RoboDK station: palletizing test.rdk

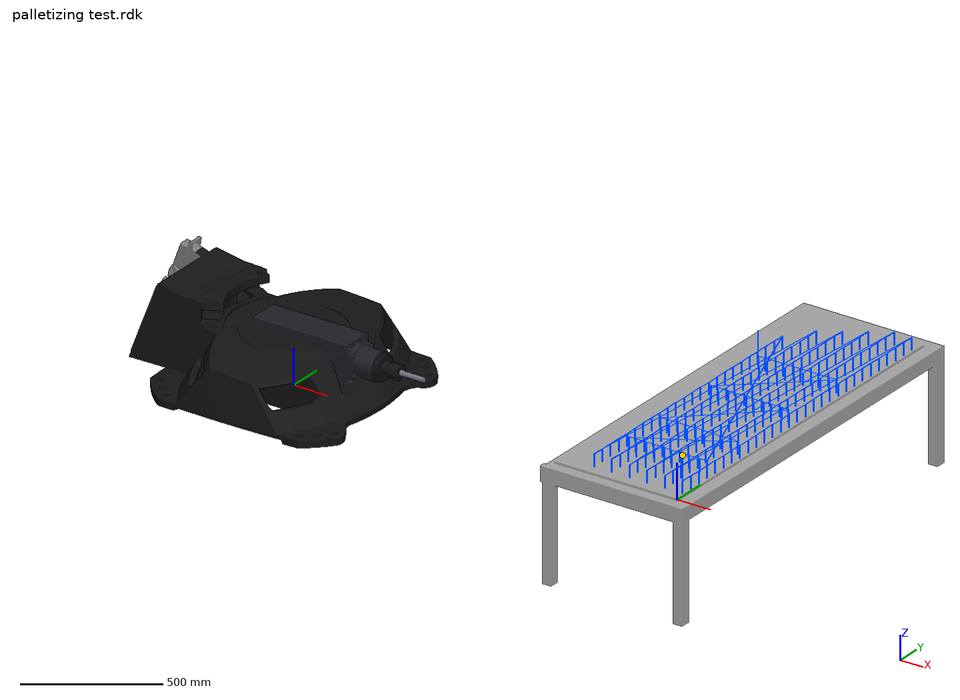
[picture v0: the station drawn from its stored meshes, robots at their saved joint values, targets as dots, program paths as lines]
Station palletizing test (saved by RoboDK 5.2.3). Poses are relative to the parent item; angles as X-Y-Z fixed-axis rotations.
  - frame KUKA KR 210 R2700 extra Base at (0, 0, 0) mm
    - robot KUKA KR 210 R2700 extra: 6 axes, payload 210 kg, reach 2696 mm, repeatability 0.06 mm, weight 1068 kg
        joint limits [-185, -140, -120, -350, -125, -350] to [185, -5, 155, 350, 125, 350]; home [0, -90, 90, 0, 0, 0]; saved at [8.498, -74.192, 109.038, -165.345, 35.74, 168.016]
      - tool Spindle, TCP at (557.2, 0, 176) mm, rotated rx 0 ry 90 rz 0 deg, size 692.9 x 170 x 256 mm
  - object Table at (1640, -780, 0) mm, size 610 x 1605 x 465 mm
  - frame Corner table at (2160, -745, 455) mm
  - object sheet c1 at (1960, 5, 455.8) mm, rotated rx 180 ry 0 rz 90 deg, size 1500 x 400 x 0.8 mm, geometry from sheet c1.stl
  - object test_multiple_points at (2160, -745, 455) mm
  - machining project Path1 settings: rotZ(0) | rotX(0)*rotY(0) | rotz(0) | onStart | onPathStart | onApproach | onPoint | onRetract | onFinish | SetRPM(%1) | SetTool(%1) | Extruder(%1) | default | default | OutOnMov(%1) | OutOffMov(%1) | onPathFinish | M_RunCode(%1)
  - program Path1 (621 instructions, listed below)
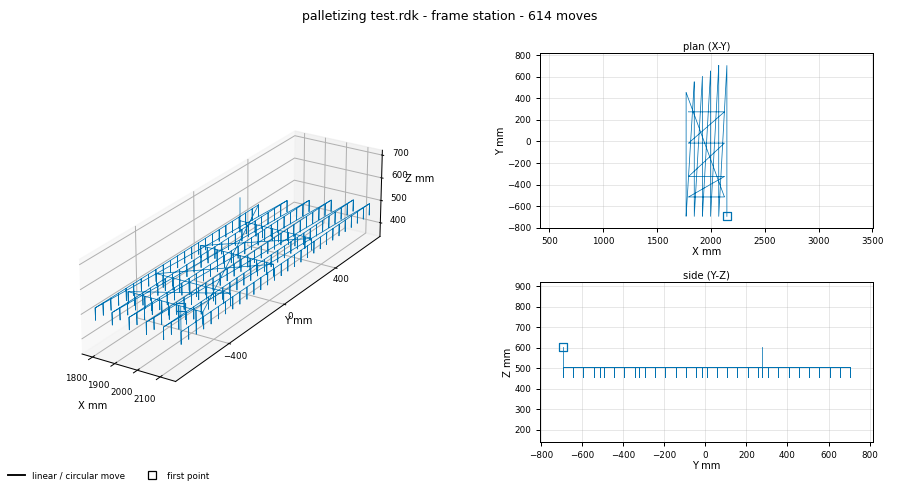
[picture p0: tool path of palletizing test.rdk in frame station, 614 of 614 moves have a stored position in this frame; points joined in program order, loops and branches not executed]

--- program Path1 (robot KUKA KR 210 R2700 extra) ---
  Smooth(1)
  Set speed (1000.0 mm/s)
  Set Ref.: Corner table
  Set Tool: Spindle
  Show Spindle
  MoveJ 1 to (-10.8, 50, 150) mm, rotated rx -180 ry 0 rz -180 deg; joints [21.568, -65.448, 91.228, -137.733, 33.132, 142.725]
  MoveL 2 to (-10.8, 50, 150) mm, rotated rx -180 ry 0 rz -180 deg; joints [21.568, -65.448, 91.228, -137.733, 33.132, 142.725]
  MoveL 3 to (-10.8, 50, 50) mm, rotated rx 180 ry 0 rz 180 deg; joints [21.568, -62.958, 93.047, -141.745, 36.422, 147.607]
  MoveL 4 to (-10.8, 50, 50) mm, rotated rx 180 ry 0 rz 180 deg; joints [21.568, -62.958, 93.047, -141.745, 36.422, 147.607]
  Set speed (50.0 mm/s)
  MoveL 5 to (-10.8, 50, -0.5) mm, rotated rx -180 ry 0 rz -180 deg; joints [21.568, -61.578, 93.809, -143.455, 38.124, 149.755]
  MoveL 6 to (-10.8, 50, 50) mm, rotated rx 180 ry 0 rz 180 deg; joints [21.568, -62.958, 93.047, -141.745, 36.422, 147.607]
  MoveL 7 to (-10.8, 100, 50) mm, rotated rx 180 ry 0 rz 180 deg; joints [20.146, -63.712, 94.184, -144.117, 35.987, 149.657]
  MoveL 8 to (-10.8, 100, -0.5) mm, rotated rx -180 ry 0 rz -180 deg; joints [20.146, -62.314, 94.947, -145.773, 37.757, 151.726]
  MoveL 9 to (-10.8, 100, 50) mm, rotated rx 180 ry 0 rz 180 deg; joints [20.146, -63.712, 94.184, -144.117, 35.987, 149.657]
  MoveL 10 to (-10.8, 150, 50) mm, rotated rx 180 ry 0 rz -180 deg; joints [18.697, -64.415, 95.236, -146.555, 35.565, 151.751]
  MoveL 11 to (-10.8, 150, -0.5) mm, rotated rx -180 ry 0 rz 180 deg; joints [18.697, -63, 96.001, -148.145, 37.401, 153.729]
  MoveL 12 to (-10.8, 150, 50) mm, rotated rx 180 ry 0 rz -180 deg; joints [18.697, -64.415, 95.236, -146.555, 35.565, 151.751]
  MoveL 13 to (-10.8, 200, 50) mm, rotated rx -180 ry 0 rz -180 deg; joints [17.222, -65.065, 96.203, -149.059, 35.16, 153.891]
  MoveL 14 to (-10.8, 200, -0.5) mm, rotated rx 180 ry 0 rz 180 deg; joints [17.222, -63.636, 96.97, -150.574, 37.059, 155.765]
  MoveL 15 to (-10.8, 200, 50) mm, rotated rx -180 ry 0 rz -180 deg; joints [17.222, -65.065, 96.203, -149.059, 35.16, 153.891]
  MoveL 16 to (-10.8, 250, 50) mm, rotated rx -180 ry 0 rz -180 deg; joints [15.724, -65.663, 97.086, -151.63, 34.774, 156.079]
  MoveL 17 to (-10.8, 250, -0.5) mm, rotated rx -180 ry 0 rz -180 deg; joints [15.724, -64.219, 97.855, -153.057, 36.734, 157.837]
  MoveL 18 to (-10.8, 250, 50) mm, rotated rx -180 ry 0 rz -180 deg; joints [15.724, -65.663, 97.086, -151.63, 34.774, 156.079]
  MoveL 19 to (-10.8, 300, 50) mm, rotated rx -180 ry 0 rz 180 deg; joints [14.203, -66.207, 97.884, -154.267, 34.411, 158.316]
  MoveL 20 to (-10.8, 300, -0.5) mm, rotated rx -180 ry 0 rz -180 deg; joints [14.203, -64.75, 98.655, -155.595, 36.43, 159.945]
  MoveL 21 to (-10.8, 300, 50) mm, rotated rx -180 ry 0 rz 180 deg; joints [14.203, -66.207, 97.884, -154.267, 34.411, 158.316]
  MoveL 22 to (-10.8, 350, 50) mm, rotated rx -180 ry 0 rz -180 deg; joints [12.662, -66.696, 98.598, -156.969, 34.075, 160.602]
  MoveL 23 to (-10.8, 350, -0.5) mm, rotated rx 180 ry 0 rz -180 deg; joints [12.662, -65.227, 99.371, -158.185, 36.148, 162.088]
  MoveL 24 to (-10.8, 350, 50) mm, rotated rx -180 ry 0 rz -180 deg; joints [12.662, -66.696, 98.598, -156.969, 34.075, 160.602]
  MoveL 25 to (-10.8, 400, 50) mm, rotated rx 180 ry 0 rz 180 deg; joints [11.102, -67.129, 99.228, -159.732, 33.77, 162.935]
  MoveL 26 to (-10.8, 400, -0.5) mm, rotated rx 180 ry 0 rz 180 deg; joints [11.102, -65.649, 100.002, -160.826, 35.891, 164.267]
  MoveL 27 to (-10.8, 400, 50) mm, rotated rx 180 ry 0 rz 180 deg; joints [11.102, -67.129, 99.228, -159.732, 33.77, 162.935]
  MoveL 28 to (-10.8, 450, 50) mm, rotated rx -180 ry 0 rz -180 deg; joints [9.525, -67.506, 99.773, -162.553, 33.497, 165.314]
  MoveL 29 to (-10.8, 450, -0.5) mm, rotated rx 180 ry 0 rz 180 deg; joints [9.525, -66.017, 100.548, -163.512, 35.663, 166.478]
  MoveL 30 to (-10.8, 450, 50) mm, rotated rx -180 ry 0 rz -180 deg; joints [9.525, -67.506, 99.773, -162.553, 33.497, 165.314]
  MoveL 31 to (-10.8, 500, 50) mm, rotated rx -180 ry 0 rz -180 deg; joints [7.933, -67.825, 100.233, -165.425, 33.261, 167.734]
  MoveL 32 to (-10.8, 500, -0.5) mm, rotated rx 180 ry 0 rz 180 deg; joints [7.933, -66.328, 101.01, -166.24, 35.466, 168.72]
  MoveL 33 to (-10.8, 500, 50) mm, rotated rx -180 ry 0 rz -180 deg; joints [7.933, -67.825, 100.233, -165.425, 33.261, 167.734]
  MoveL 34 to (-10.8, 550, 50) mm, rotated rx 180 ry 0 rz 180 deg; joints [6.329, -68.086, 100.608, -168.344, 33.065, 170.191]
  MoveL 35 to (-10.8, 550, -0.5) mm, rotated rx 180 ry 0 rz 180 deg; joints [6.329, -66.583, 101.386, -169.003, 35.302, 170.989]
  MoveL 36 to (-10.8, 550, 50) mm, rotated rx 180 ry 0 rz 180 deg; joints [6.329, -68.086, 100.608, -168.344, 33.065, 170.191]
  MoveL 37 to (-10.8, 600, 50) mm, rotated rx -180 ry 0 rz -180 deg; joints [4.715, -68.289, 100.897, -171.299, 32.911, 172.679]
  MoveL 38 to (-10.8, 600, -0.5) mm, rotated rx 180 ry 0 rz 180 deg; joints [4.715, -66.78, 101.677, -171.797, 35.174, 173.28]
  MoveL 39 to (-10.8, 600, 50) mm, rotated rx -180 ry 0 rz -180 deg; joints [4.715, -68.289, 100.897, -171.299, 32.911, 172.679]
  MoveL 40 to (-10.8, 650, 50) mm, rotated rx -180 ry 0 rz -180 deg; joints [3.093, -68.432, 101.102, -174.284, 32.8, 175.191]
  MoveL 41 to (-10.8, 650, -0.5) mm, rotated rx -180 ry 0 rz 180 deg; joints [3.093, -66.92, 101.882, -174.613, 35.082, 175.588]
  MoveL 42 to (-10.8, 650, 50) mm, rotated rx -180 ry 0 rz -180 deg; joints [3.093, -68.432, 101.102, -174.284, 32.8, 175.191]
  MoveL 43 to (-10.8, 700, 50) mm, rotated rx 180 ry 0 rz 180 deg; joints [1.466, -68.516, 101.222, -177.288, 32.735, 177.718]
  MoveL 44 to (-10.8, 700, -0.5) mm, rotated rx -180 ry 0 rz -180 deg; joints [1.466, -67.001, 102.002, -177.445, 35.028, 177.907]
  MoveL 45 to (-10.8, 700, 50) mm, rotated rx 180 ry 0 rz 180 deg; joints [1.466, -68.516, 101.222, -177.288, 32.735, 177.718]
  MoveL 46 to (-10.8, 750, 50) mm, rotated rx -180 ry 0 rz -180 deg; joints [-0.163, -68.54, 101.256, -180.301, 32.717, 180.254]
  MoveL 47 to (-10.8, 750, -0.5) mm, rotated rx -180 ry 0 rz -180 deg; joints [-0.163, -67.024, 102.036, -180.284, 35.012, 180.233]
  MoveL 48 to (-10.8, 750, 50) mm, rotated rx -180 ry 0 rz -180 deg; joints [-0.163, -68.54, 101.256, -180.301, 32.717, 180.254]
  MoveL 49 to (-10.8, 800, 50) mm, rotated rx -180 ry 0 rz -180 deg; joints [-1.792, -68.504, 101.205, -183.314, 32.745, 182.788]
  MoveL 50 to (-10.8, 800, -0.5) mm, rotated rx 180 ry 0 rz -180 deg; joints [-1.792, -66.989, 101.985, -183.122, 35.035, 182.557]
  MoveL 51 to (-10.8, 800, 50) mm, rotated rx -180 ry 0 rz -180 deg; joints [-1.792, -68.504, 101.205, -183.314, 32.745, 182.788]
  MoveL 52 to (-10.8, 850, 50) mm, rotated rx 180 ry 0 rz 180 deg; joints [-3.418, -68.408, 101.068, -186.315, 32.819, 185.313]
  MoveL 53 to (-10.8, 850, -0.5) mm, rotated rx 180 ry 0 rz -180 deg; joints [-3.418, -66.896, 101.848, -185.951, 35.097, 184.875]
  MoveL 54 to (-10.8, 850, 50) mm, rotated rx 180 ry 0 rz 180 deg; joints [-3.418, -68.408, 101.068, -186.315, 32.819, 185.313]
  MoveL 55 to (-10.8, 900, 50) mm, rotated rx 180 ry 0 rz 180 deg; joints [-5.038, -68.253, 100.846, -189.295, 32.938, 187.821]
  MoveL 56 to (-10.8, 900, -0.5) mm, rotated rx -180 ry 0 rz -180 deg; joints [-5.038, -66.745, 101.625, -188.764, 35.197, 187.18]
  MoveL 57 to (-10.8, 900, 50) mm, rotated rx 180 ry 0 rz 180 deg; joints [-5.038, -68.253, 100.846, -189.295, 32.938, 187.821]
  MoveL 58 to (-10.8, 950, 50) mm, rotated rx -180 ry 0 rz -180 deg; joints [-6.65, -68.039, 100.539, -192.243, 33.101, 190.303]
  MoveL 59 to (-10.8, 950, -0.5) mm, rotated rx -180 ry 0 rz -180 deg; joints [-6.65, -66.536, 101.317, -191.552, 35.333, 189.467]
  MoveL 60 to (-10.8, 950, 50) mm, rotated rx -180 ry 0 rz -180 deg; joints [-6.65, -68.039, 100.539, -192.243, 33.101, 190.303]
  MoveL 61 to (-10.8, 1000, 50) mm, rotated rx -180 ry 0 rz -180 deg; joints [-8.252, -67.766, 100.147, -195.153, 33.305, 192.753]
  MoveL 62 to (-10.8, 1000, -0.5) mm, rotated rx -180 ry 0 rz -180 deg; joints [-8.252, -66.27, 100.924, -194.309, 35.503, 191.73]
  MoveL 63 to (-10.8, 1000, 50) mm, rotated rx -180 ry 0 rz -180 deg; joints [-8.252, -67.766, 100.147, -195.153, 33.305, 192.753]
  MoveL 64 to (-10.8, 1050, 50) mm, rotated rx -180 ry 0 rz -180 deg; joints [-9.841, -67.435, 99.67, -198.016, 33.549, 195.165]
  MoveL 65 to (-10.8, 1050, -0.5) mm, rotated rx -180 ry 0 rz -180 deg; joints [-9.841, -65.948, 100.446, -197.029, 35.707, 193.966]
  MoveL 66 to (-10.8, 1050, 50) mm, rotated rx -180 ry 0 rz -180 deg; joints [-9.841, -67.435, 99.67, -198.016, 33.549, 195.165]
  MoveL 67 to (-10.8, 1100, 50) mm, rotated rx -180 ry 0 rz -180 deg; joints [-11.415, -67.047, 99.109, -200.825, 33.828, 197.535]
  MoveL 68 to (-10.8, 1100, -0.5) mm, rotated rx -180 ry 0 rz -180 deg; joints [-11.415, -65.569, 99.883, -199.706, 35.941, 196.172]
  MoveL 69 to (-10.8, 1100, 50) mm, rotated rx -180 ry 0 rz -180 deg; joints [-11.415, -67.047, 99.109, -200.825, 33.828, 197.535]
  MoveL 70 to (-10.8, 1150, 50) mm, rotated rx 180 ry 0 rz -180 deg; joints [-12.972, -66.602, 98.462, -203.576, 34.14, 199.859]
  MoveL 71 to (-10.8, 1150, -0.5) mm, rotated rx 180 ry 0 rz -180 deg; joints [-12.972, -65.136, 99.235, -202.337, 36.202, 198.343]
  MoveL 72 to (-10.8, 1150, 50) mm, rotated rx 180 ry 0 rz -180 deg; joints [-12.972, -66.602, 98.462, -203.576, 34.14, 199.859]
  MoveL 73 to (-10.8, 1200, 50) mm, rotated rx 180 ry 0 rz -180 deg; joints [-14.509, -66.102, 97.732, -206.265, 34.482, 202.135]
  MoveL 74 to (-10.8, 1200, -0.5) mm, rotated rx 180 ry 0 rz -180 deg; joints [-14.509, -64.648, 98.502, -204.917, 36.489, 200.48]
  MoveL 75 to (-10.8, 1200, 50) mm, rotated rx 180 ry 0 rz -180 deg; joints [-14.509, -66.102, 97.732, -206.265, 34.482, 202.135]
  MoveL 76 to (-10.8, 1250, 50) mm, rotated rx 180 ry 0 rz -180 deg; joints [-16.025, -65.548, 96.916, -208.889, 34.849, 204.362]
  MoveL 77 to (-10.8, 1250, -0.5) mm, rotated rx -180 ry 0 rz -180 deg; joints [-16.025, -64.106, 97.685, -207.444, 36.798, 202.58]
  MoveL 78 to (-10.8, 1250, 50) mm, rotated rx 180 ry 0 rz -180 deg; joints [-16.025, -65.548, 96.916, -208.889, 34.849, 204.362]
  MoveL 79 to (-10.8, 1300, 50) mm, rotated rx -180 ry 0 rz -180 deg; joints [-17.519, -64.94, 96.016, -211.447, 35.239, 206.541]
  MoveL 80 to (-10.8, 1300, -0.5) mm, rotated rx 180 ry 0 rz 180 deg; joints [-17.519, -63.513, 96.783, -209.917, 37.126, 204.645]
  MoveL 81 to (-10.8, 1300, 50) mm, rotated rx -180 ry 0 rz -180 deg; joints [-17.519, -64.94, 96.016, -211.447, 35.239, 206.541]
  MoveL 82 to (-10.8, 1350, 50) mm, rotated rx 180 ry 0 rz -180 deg; joints [-18.988, -64.279, 95.032, -213.938, 35.648, 208.671]
  MoveL 83 to (-10.8, 1350, -0.5) mm, rotated rx -180 ry 0 rz -180 deg; joints [-18.988, -62.867, 95.797, -212.334, 37.471, 206.674]
  MoveL 84 to (-10.8, 1350, 50) mm, rotated rx 180 ry 0 rz -180 deg; joints [-18.988, -64.279, 95.032, -213.938, 35.648, 208.671]
  MoveL 85 to (-10.8, 1400, 50) mm, rotated rx 180 ry 0 rz 180 deg; joints [-20.432, -63.566, 93.963, -216.362, 36.073, 210.756]
  MoveL 86 to (-10.8, 1400, -0.5) mm, rotated rx 180 ry 0 rz -180 deg; joints [-20.432, -62.171, 94.726, -214.695, 37.829, 208.67]
  MoveL 87 to (-10.8, 1400, 50) mm, rotated rx 180 ry 0 rz 180 deg; joints [-20.432, -63.566, 93.963, -216.362, 36.073, 210.756]
  MoveL 88 to (-10.8, 1450, 50) mm, rotated rx 180 ry 0 rz 180 deg; joints [-21.85, -62.802, 92.809, -218.722, 36.51, 212.799]
  MoveL 89 to (-10.8, 1450, -0.5) mm, rotated rx 180 ry 0 rz -180 deg; joints [-21.85, -61.424, 93.571, -217.002, 38.199, 210.635]
  MoveL 90 to (-10.8, 1450, 50) mm, rotated rx 180 ry 0 rz 180 deg; joints [-21.85, -62.802, 92.809, -218.722, 36.51, 212.799]
  MoveL 91 to (-86.48, 50, 50) mm, rotated rx 180 ry 0 rz 180 deg; joints [22.444, -65.922, 97.466, -141.707, 38.031, 148.122]
  MoveL 92 to (-86.48, 50, -0.5) mm, rotated rx 180 ry 0 rz 180 deg; joints [22.444, -64.471, 98.236, -143.379, 39.794, 150.271]
  MoveL 93 to (-86.48, 50, 50) mm, rotated rx 180 ry 0 rz 180 deg; joints [22.444, -65.922, 97.466, -141.707, 38.031, 148.122]
  MoveL 94 to (-86.48, 100, 50) mm, rotated rx -180 ry 0 rz -180 deg; joints [20.975, -66.7, 98.605, -144.045, 37.564, 150.102]
  MoveL 95 to (-86.48, 100, -0.5) mm, rotated rx -180 ry 0 rz -180 deg; joints [20.975, -65.231, 99.378, -145.668, 39.397, 152.176]
  MoveL 96 to (-86.48, 100, 50) mm, rotated rx -180 ry 0 rz -180 deg; joints [20.975, -66.7, 98.605, -144.045, 37.564, 150.102]
  MoveL 97 to (-86.48, 150, 50) mm, rotated rx -180 ry 0 rz -180 deg; joints [19.475, -67.428, 99.66, -146.454, 37.109, 152.131]
  MoveL 98 to (-86.48, 150, -0.5) mm, rotated rx -180 ry 0 rz 180 deg; joints [19.475, -65.941, 100.436, -148.018, 39.011, 154.118]
  MoveL 99 to (-86.48, 150, 50) mm, rotated rx -180 ry 0 rz -180 deg; joints [19.475, -67.428, 99.66, -146.454, 37.109, 152.131]
  MoveL 100 to (-86.48, 200, 50) mm, rotated rx 180 ry 0 rz 180 deg; joints [17.948, -68.103, 100.631, -148.936, 36.67, 154.211]
  MoveL 101 to (-86.48, 200, -0.5) mm, rotated rx 180 ry 0 rz 180 deg; joints [17.948, -66.599, 101.41, -150.429, 38.64, 156.097]
  MoveL 102 to (-86.48, 200, 50) mm, rotated rx 180 ry 0 rz 180 deg; joints [17.948, -68.103, 100.631, -148.936, 36.67, 154.211]
  MoveL 103 to (-86.48, 250, 50) mm, rotated rx -180 ry 0 rz -180 deg; joints [16.394, -68.724, 101.519, -151.49, 36.25, 156.345]
  MoveL 104 to (-86.48, 250, -0.5) mm, rotated rx 180 ry 0 rz 180 deg; joints [16.394, -67.204, 102.3, -152.901, 38.286, 158.117]
  MoveL 105 to (-86.48, 250, 50) mm, rotated rx -180 ry 0 rz -180 deg; joints [16.394, -68.724, 101.519, -151.49, 36.25, 156.345]
  MoveL 106 to (-86.48, 300, 50) mm, rotated rx -180 ry 0 rz -180 deg; joints [14.815, -69.29, 102.322, -154.117, 35.855, 158.532]
  MoveL 107 to (-86.48, 300, -0.5) mm, rotated rx -180 ry 0 rz -180 deg; joints [14.815, -67.756, 103.106, -155.433, 37.952, 160.178]
  MoveL 108 to (-86.48, 300, 50) mm, rotated rx -180 ry 0 rz -180 deg; joints [14.815, -69.29, 102.322, -154.117, 35.855, 158.532]
  MoveL 109 to (-86.48, 350, 50) mm, rotated rx 180 ry 0 rz -180 deg; joints [13.212, -69.801, 103.041, -156.815, 35.487, 160.775]
  MoveL 110 to (-86.48, 350, -0.5) mm, rotated rx 180 ry 0 rz 180 deg; joints [13.212, -68.253, 103.827, -158.024, 37.643, 162.279]
  MoveL 111 to (-86.48, 350, 50) mm, rotated rx 180 ry 0 rz -180 deg; joints [13.212, -69.801, 103.041, -156.815, 35.487, 160.775]
  MoveL 112 to (-86.48, 400, 50) mm, rotated rx 180 ry 0 rz -180 deg; joints [11.588, -70.253, 103.675, -159.581, 35.152, 163.07]
  MoveL 113 to (-86.48, 400, -0.5) mm, rotated rx 180 ry 0 rz 180 deg; joints [11.588, -68.694, 104.464, -160.669, 37.36, 164.42]
  MoveL 114 to (-86.48, 400, 50) mm, rotated rx 180 ry 0 rz -180 deg; joints [11.588, -70.253, 103.675, -159.581, 35.152, 163.07]
  MoveL 115 to (-86.48, 450, 50) mm, rotated rx -180 ry 0 rz -180 deg; joints [9.945, -70.648, 104.224, -162.41, 34.852, 165.417]
  MoveL 116 to (-86.48, 450, -0.5) mm, rotated rx 180 ry 0 rz 180 deg; joints [9.945, -69.078, 105.016, -163.367, 37.109, 166.599]
  MoveL 117 to (-86.48, 450, 50) mm, rotated rx -180 ry 0 rz -180 deg; joints [9.945, -70.648, 104.224, -162.41, 34.852, 165.417]
  MoveL 118 to (-86.48, 500, 50) mm, rotated rx 180 ry 0 rz 180 deg; joints [8.285, -70.982, 104.688, -165.297, 34.592, 167.811]
  MoveL 119 to (-86.48, 500, -0.5) mm, rotated rx -180 ry 0 rz -180 deg; joints [8.285, -69.404, 105.482, -166.111, 36.891, 168.813]
  MoveL 120 to (-86.48, 500, 50) mm, rotated rx 180 ry 0 rz 180 deg; joints [8.285, -70.982, 104.688, -165.297, 34.592, 167.811]
  MoveL 121 to (-86.48, 550, 50) mm, rotated rx 180 ry 0 rz -180 deg; joints [6.611, -71.256, 105.067, -168.235, 34.375, 170.246]
  MoveL 122 to (-86.48, 550, -0.5) mm, rotated rx 180 ry 0 rz 180 deg; joints [6.611, -69.671, 105.862, -168.895, 36.709, 171.058]
  MoveL 123 to (-86.48, 550, 50) mm, rotated rx 180 ry 0 rz -180 deg; joints [6.611, -71.256, 105.067, -168.235, 34.375, 170.246]
  MoveL 124 to (-86.48, 600, 50) mm, rotated rx 180 ry 0 rz 180 deg; joints [4.926, -71.469, 105.36, -171.214, 34.205, 172.716]
  MoveL 125 to (-86.48, 600, -0.5) mm, rotated rx -180 ry 0 rz -180 deg; joints [4.926, -69.877, 106.156, -171.713, 36.566, 173.328]
  MoveL 126 to (-86.48, 600, 50) mm, rotated rx 180 ry 0 rz 180 deg; joints [4.926, -71.469, 105.36, -171.214, 34.205, 172.716]
  MoveL 127 to (-86.48, 650, 50) mm, rotated rx 180 ry 0 rz 180 deg; joints [3.232, -71.619, 105.566, -174.226, 34.082, 175.213]
  MoveL 128 to (-86.48, 650, -0.5) mm, rotated rx -180 ry 0 rz -180 deg; joints [3.232, -70.024, 106.363, -174.557, 36.463, 175.618]
  MoveL 129 to (-86.48, 650, 50) mm, rotated rx 180 ry 0 rz 180 deg; joints [3.232, -71.619, 105.566, -174.226, 34.082, 175.213]
  MoveL 130 to (-86.48, 700, 50) mm, rotated rx -180 ry 0 rz 180 deg; joints [1.532, -71.707, 105.687, -177.26, 34.01, 177.728]
  MoveL 131 to (-86.48, 700, -0.5) mm, rotated rx 180 ry 0 rz -180 deg; joints [1.532, -70.109, 106.485, -177.418, 36.403, 177.921]
  MoveL 132 to (-86.48, 700, 50) mm, rotated rx -180 ry 0 rz 180 deg; joints [1.532, -71.707, 105.687, -177.26, 34.01, 177.728]
  MoveL 133 to (-86.48, 750, 50) mm, rotated rx -180 ry 0 rz -180 deg; joints [-0.17, -71.732, 105.722, -180.305, 33.99, 180.253]
  MoveL 134 to (-86.48, 750, -0.5) mm, rotated rx 180 ry 0 rz -180 deg; joints [-0.17, -70.134, 106.519, -180.287, 36.386, 180.231]
  MoveL 135 to (-86.48, 750, 50) mm, rotated rx -180 ry 0 rz -180 deg; joints [-0.17, -71.732, 105.722, -180.305, 33.99, 180.253]
  MoveL 136 to (-86.48, 800, 50) mm, rotated rx 180 ry 0 rz -180 deg; joints [-1.872, -71.694, 105.67, -183.348, 34.021, 182.776]
  MoveL 137 to (-86.48, 800, -0.5) mm, rotated rx 180 ry 0 rz 180 deg; joints [-1.872, -70.097, 106.467, -183.155, 36.412, 182.54]
  MoveL 138 to (-86.48, 800, 50) mm, rotated rx 180 ry 0 rz -180 deg; joints [-1.872, -71.694, 105.67, -183.348, 34.021, 182.776]
  MoveL 139 to (-86.48, 850, 50) mm, rotated rx -180 ry 0 rz -180 deg; joints [-3.571, -71.594, 105.532, -186.378, 34.103, 185.288]
  MoveL 140 to (-86.48, 850, -0.5) mm, rotated rx -180 ry 0 rz -180 deg; joints [-3.571, -69.999, 106.329, -186.013, 36.48, 184.841]
  MoveL 141 to (-86.48, 850, 50) mm, rotated rx -180 ry 0 rz -180 deg; joints [-3.571, -71.594, 105.532, -186.378, 34.103, 185.288]
  MoveL 142 to (-86.48, 900, 50) mm, rotated rx -180 ry 0 rz -180 deg; joints [-5.263, -71.431, 105.308, -189.384, 34.235, 187.78]
  MoveL 143 to (-86.48, 900, -0.5) mm, rotated rx 180 ry 0 rz -180 deg; joints [-5.263, -69.841, 106.104, -188.853, 36.591, 187.128]
  MoveL 144 to (-86.48, 900, 50) mm, rotated rx -180 ry 0 rz -180 deg; joints [-5.263, -71.431, 105.308, -189.384, 34.235, 187.78]
  MoveL 145 to (-86.48, 950, 50) mm, rotated rx 180 ry 0 rz -180 deg; joints [-6.947, -71.206, 104.998, -192.357, 34.415, 190.244]
  MoveL 146 to (-86.48, 950, -0.5) mm, rotated rx -180 ry 0 rz -180 deg; joints [-6.947, -69.622, 105.793, -191.664, 36.742, 189.393]
  MoveL 147 to (-86.48, 950, 50) mm, rotated rx 180 ry 0 rz -180 deg; joints [-6.947, -71.206, 104.998, -192.357, 34.415, 190.244]
  MoveL 148 to (-86.48, 1000, 50) mm, rotated rx 180 ry 0 rz 180 deg; joints [-8.618, -70.92, 104.602, -195.285, 34.641, 192.671]
  MoveL 149 to (-86.48, 1000, -0.5) mm, rotated rx -180 ry 0 rz -180 deg; joints [-8.618, -69.343, 105.395, -194.441, 36.931, 191.632]
  MoveL 150 to (-86.48, 1000, 50) mm, rotated rx 180 ry 0 rz 180 deg; joints [-8.618, -70.92, 104.602, -195.285, 34.641, 192.671]
  MoveL 151 to (-86.48, 1050, 50) mm, rotated rx -180 ry 0 rz -180 deg; joints [-10.275, -70.573, 104.121, -198.161, 34.909, 195.056]
  MoveL 152 to (-86.48, 1050, -0.5) mm, rotated rx -180 ry 0 rz -180 deg; joints [-10.275, -69.006, 104.912, -197.176, 37.156, 193.839]
  MoveL 153 to (-86.48, 1050, 50) mm, rotated rx -180 ry 0 rz -180 deg; joints [-10.275, -70.573, 104.121, -198.161, 34.909, 195.056]
  MoveL 154 to (-86.48, 1100, 50) mm, rotated rx 180 ry 0 rz -180 deg; joints [-11.914, -70.167, 103.555, -200.978, 35.216, 197.393]
  MoveL 155 to (-86.48, 1100, -0.5) mm, rotated rx -180 ry 0 rz -180 deg; joints [-11.914, -68.611, 104.344, -199.864, 37.415, 196.011]
  MoveL 156 to (-86.48, 1100, 50) mm, rotated rx 180 ry 0 rz -180 deg; joints [-11.914, -70.167, 103.555, -200.978, 35.216, 197.393]
  MoveL 157 to (-86.48, 1150, 50) mm, rotated rx 180 ry 0 rz -180 deg; joints [-13.534, -69.703, 102.904, -203.73, 35.559, 199.678]
  MoveL 158 to (-86.48, 1150, -0.5) mm, rotated rx 180 ry 0 rz 180 deg; joints [-13.534, -68.158, 103.69, -202.499, 37.703, 198.144]
  MoveL 159 to (-86.48, 1150, 50) mm, rotated rx 180 ry 0 rz -180 deg; joints [-13.534, -69.703, 102.904, -203.73, 35.559, 199.678]
  MoveL 160 to (-86.48, 1200, 50) mm, rotated rx 180 ry 0 rz -180 deg; joints [-15.132, -69.182, 102.168, -206.414, 35.932, 201.91]
  MoveL 161 to (-86.48, 1200, -0.5) mm, rotated rx 180 ry 0 rz 180 deg; joints [-15.132, -67.65, 102.951, -205.078, 38.017, 200.238]
  MoveL 162 to (-86.48, 1200, 50) mm, rotated rx 180 ry 0 rz -180 deg; joints [-15.132, -69.182, 102.168, -206.414, 35.932, 201.91]
  MoveL 163 to (-86.48, 1250, 50) mm, rotated rx 180 ry 0 rz 180 deg; joints [-16.707, -68.604, 101.348, -209.027, 36.332, 204.086]
  MoveL 164 to (-86.48, 1250, -0.5) mm, rotated rx 180 ry 0 rz 180 deg; joints [-16.707, -67.087, 102.129, -207.598, 38.355, 202.29]
  MoveL 165 to (-86.48, 1250, 50) mm, rotated rx 180 ry 0 rz 180 deg; joints [-16.707, -68.604, 101.348, -209.027, 36.332, 204.086]
  MoveL 166 to (-86.48, 1300, 50) mm, rotated rx 180 ry 0 rz -180 deg; joints [-18.256, -67.972, 100.444, -211.567, 36.756, 206.209]
  MoveL 167 to (-86.48, 1300, -0.5) mm, rotated rx 180 ry 0 rz 180 deg; joints [-18.256, -66.471, 101.222, -210.058, 38.713, 204.302]
  MoveL 168 to (-86.48, 1300, 50) mm, rotated rx 180 ry 0 rz -180 deg; joints [-18.256, -67.972, 100.444, -211.567, 36.756, 206.209]
  MoveL 169 to (-86.48, 1350, 50) mm, rotated rx 180 ry 0 rz -180 deg; joints [-19.778, -67.286, 99.456, -214.034, 37.198, 208.278]
  MoveL 170 to (-86.48, 1350, -0.5) mm, rotated rx 180 ry 0 rz -180 deg; joints [-19.778, -65.803, 100.231, -212.457, 39.088, 206.274]
  MoveL 171 to (-86.48, 1350, 50) mm, rotated rx 180 ry 0 rz -180 deg; joints [-19.778, -67.286, 99.456, -214.034, 37.198, 208.278]
  MoveL 172 to (-86.48, 1400, 50) mm, rotated rx 180 ry 0 rz -180 deg; joints [-21.271, -66.549, 98.384, -216.428, 37.656, 210.297]
  MoveL 173 to (-86.48, 1400, -0.5) mm, rotated rx 180 ry 0 rz 180 deg; joints [-21.271, -65.083, 99.156, -214.794, 39.475, 208.208]
  MoveL 174 to (-86.48, 1400, 50) mm, rotated rx 180 ry 0 rz -180 deg; joints [-21.271, -66.549, 98.384, -216.428, 37.656, 210.297]
  MoveL 175 to (-86.48, 1450, 50) mm, rotated rx -180 ry 0 rz -180 deg; joints [-22.734, -65.76, 97.229, -218.753, 38.126, 212.269]
  MoveL 176 to (-86.48, 1450, -0.5) mm, rotated rx 180 ry 0 rz -180 deg; joints [-22.734, -64.313, 97.998, -217.071, 39.874, 210.106]
  MoveL 177 to (-86.48, 1450, 50) mm, rotated rx -180 ry 0 rz -180 deg; joints [-22.734, -65.76, 97.229, -218.753, 38.126, 212.269]
  MoveL 178 to (-162.16, 50, 50) mm, rotated rx -180 ry 0 rz -180 deg; joints [23.39, -68.855, 101.705, -141.432, 39.551, 148.416]
  MoveL 179 to (-162.16, 50, -0.5) mm, rotated rx 180 ry 0 rz -180 deg; joints [23.39, -67.332, 102.487, -143.087, 41.374, 150.59]
  MoveL 180 to (-162.16, 50, 50) mm, rotated rx -180 ry 0 rz -180 deg; joints [23.39, -68.855, 101.705, -141.432, 39.551, 148.416]
  MoveL 181 to (-162.16, 100, 50) mm, rotated rx -180 ry 0 rz 180 deg; joints [21.871, -69.666, 102.851, -143.745, 39.044, 150.335]
  MoveL 182 to (-162.16, 100, -0.5) mm, rotated rx 180 ry 0 rz -180 deg; joints [21.871, -68.122, 103.637, -145.356, 40.942, 152.437]
  MoveL 183 to (-162.16, 100, 50) mm, rotated rx -180 ry 0 rz 180 deg; joints [21.871, -69.666, 102.851, -143.745, 39.044, 150.335]
  MoveL 184 to (-162.16, 150, 50) mm, rotated rx 180 ry 0 rz 180 deg; joints [20.319, -70.425, 103.914, -146.135, 38.548, 152.307]
  MoveL 185 to (-162.16, 150, -0.5) mm, rotated rx -180 ry 0 rz -180 deg; joints [20.319, -68.861, 104.704, -147.692, 40.52, 154.326]
  MoveL 186 to (-162.16, 150, 50) mm, rotated rx 180 ry 0 rz 180 deg; joints [20.319, -70.425, 103.914, -146.135, 38.548, 152.307]
  MoveL 187 to (-162.16, 200, 50) mm, rotated rx -180 ry 0 rz -180 deg; joints [18.736, -71.131, 104.894, -148.605, 38.067, 154.337]
  MoveL 188 to (-162.16, 200, -0.5) mm, rotated rx 180 ry 0 rz -180 deg; joints [18.736, -69.548, 105.688, -150.096, 40.112, 156.258]
  MoveL 189 to (-162.16, 200, 50) mm, rotated rx -180 ry 0 rz -180 deg; joints [18.736, -71.131, 104.894, -148.605, 38.067, 154.337]
  MoveL 190 to (-162.16, 250, 50) mm, rotated rx -180 ry 0 rz -180 deg; joints [17.122, -71.782, 105.789, -151.155, 37.606, 156.426]
  MoveL 191 to (-162.16, 250, -0.5) mm, rotated rx -180 ry 0 rz 180 deg; joints [17.122, -70.182, 106.588, -152.568, 39.721, 158.236]
  MoveL 192 to (-162.16, 250, 50) mm, rotated rx -180 ry 0 rz -180 deg; joints [17.122, -71.782, 105.789, -151.155, 37.606, 156.426]
  MoveL 193 to (-162.16, 300, 50) mm, rotated rx 180 ry 0 rz 180 deg; joints [15.48, -72.377, 106.601, -153.785, 37.17, 158.577]
  MoveL 194 to (-162.16, 300, -0.5) mm, rotated rx 180 ry 0 rz 180 deg; joints [15.48, -70.761, 107.403, -155.107, 39.351, 160.261]
  MoveL 195 to (-162.16, 300, 50) mm, rotated rx 180 ry 0 rz 180 deg; joints [15.48, -72.377, 106.601, -153.785, 37.17, 158.577]
  MoveL 196 to (-162.16, 350, 50) mm, rotated rx 180 ry 0 rz 180 deg; joints [13.811, -72.913, 107.328, -156.493, 36.763, 160.789]
  MoveL 197 to (-162.16, 350, -0.5) mm, rotated rx 180 ry 0 rz -180 deg; joints [13.811, -71.283, 108.134, -157.712, 39.007, 162.333]
  MoveL 198 to (-162.16, 350, 50) mm, rotated rx 180 ry 0 rz 180 deg; joints [13.811, -72.913, 107.328, -156.493, 36.763, 160.789]
  MoveL 199 to (-162.16, 400, 50) mm, rotated rx 180 ry 0 rz 180 deg; joints [12.118, -73.391, 107.97, -159.278, 36.39, 163.063]
  MoveL 200 to (-162.16, 400, -0.5) mm, rotated rx -180 ry 0 rz -180 deg; joints [12.118, -71.747, 108.779, -160.379, 38.692, 164.45]
  MoveL 201 to (-162.16, 400, 50) mm, rotated rx 180 ry 0 rz 180 deg; joints [12.118, -73.391, 107.97, -159.278, 36.39, 163.063]
  MoveL 202 to (-162.16, 450, 50) mm, rotated rx 180 ry 0 rz 180 deg; joints [10.403, -73.807, 108.526, -162.134, 36.057, 165.394]
  MoveL 203 to (-162.16, 450, -0.5) mm, rotated rx 180 ry 0 rz 180 deg; joints [10.403, -72.152, 109.338, -163.104, 38.411, 166.612]
  MoveL 204 to (-162.16, 450, 50) mm, rotated rx 180 ry 0 rz 180 deg; joints [10.403, -73.807, 108.526, -162.134, 36.057, 165.394]
  MoveL 205 to (-162.16, 500, 50) mm, rotated rx 180 ry 0 rz -180 deg; joints [8.669, -74.16, 108.997, -165.055, 35.766, 167.78]
  MoveL 206 to (-162.16, 500, -0.5) mm, rotated rx 180 ry 0 rz 180 deg; joints [8.669, -72.496, 109.811, -165.882, 38.166, 168.814]
  MoveL 207 to (-162.16, 500, 50) mm, rotated rx 180 ry 0 rz -180 deg; joints [8.669, -74.16, 108.997, -165.055, 35.766, 167.78]
  MoveL 208 to (-162.16, 550, 50) mm, rotated rx 180 ry 0 rz 180 deg; joints [6.919, -74.45, 109.381, -168.033, 35.523, 170.213]
  MoveL 209 to (-162.16, 550, -0.5) mm, rotated rx -180 ry 0 rz -180 deg; joints [6.919, -72.778, 110.197, -168.706, 37.962, 171.052]
  MoveL 210 to (-162.16, 550, 50) mm, rotated rx 180 ry 0 rz 180 deg; joints [6.919, -74.45, 109.381, -168.033, 35.523, 170.213]
  MoveL 211 to (-162.16, 600, 50) mm, rotated rx -180 ry 0 rz -180 deg; joints [5.156, -74.675, 109.678, -171.06, 35.332, 172.686]
  MoveL 212 to (-162.16, 600, -0.5) mm, rotated rx -180 ry 0 rz 180 deg; joints [5.156, -72.996, 110.496, -171.568, 37.8, 173.319]
  MoveL 213 to (-162.16, 600, 50) mm, rotated rx -180 ry 0 rz -180 deg; joints [5.156, -74.675, 109.678, -171.06, 35.332, 172.686]
  MoveL 214 to (-162.16, 650, 50) mm, rotated rx 180 ry 0 rz -180 deg; joints [3.384, -74.835, 109.887, -174.123, 35.194, 175.191]
  MoveL 215 to (-162.16, 650, -0.5) mm, rotated rx -180 ry 0 rz -180 deg; joints [3.384, -73.152, 110.707, -174.46, 37.685, 175.61]
  MoveL 216 to (-162.16, 650, 50) mm, rotated rx 180 ry 0 rz -180 deg; joints [3.384, -74.835, 109.887, -174.123, 35.194, 175.191]
  MoveL 217 to (-162.16, 700, 50) mm, rotated rx 180 ry 0 rz 180 deg; joints [1.604, -74.928, 110.01, -177.21, 35.113, 177.717]
  MoveL 218 to (-162.16, 700, -0.5) mm, rotated rx 180 ry 0 rz 180 deg; joints [1.604, -73.242, 110.83, -177.371, 37.617, 177.917]
  MoveL 219 to (-162.16, 700, 50) mm, rotated rx 180 ry 0 rz 180 deg; joints [1.604, -74.928, 110.01, -177.21, 35.113, 177.717]
  MoveL 220 to (-162.16, 750, 50) mm, rotated rx 180 ry 0 rz -180 deg; joints [-0.178, -74.955, 110.045, -180.31, 35.09, 180.254]
  MoveL 221 to (-162.16, 750, -0.5) mm, rotated rx 180 ry 0 rz 180 deg; joints [-0.178, -73.268, 110.865, -180.292, 37.597, 180.232]
  MoveL 222 to (-162.16, 750, 50) mm, rotated rx 180 ry 0 rz -180 deg; joints [-0.178, -74.955, 110.045, -180.31, 35.09, 180.254]
  MoveL 223 to (-162.16, 800, 50) mm, rotated rx 180 ry 0 rz 180 deg; joints [-1.96, -74.915, 109.992, -183.409, 35.125, 182.789]
  MoveL 224 to (-162.16, 800, -0.5) mm, rotated rx 180 ry 0 rz -180 deg; joints [-1.96, -73.229, 110.812, -183.212, 37.627, 182.545]
  MoveL 225 to (-162.16, 800, 50) mm, rotated rx 180 ry 0 rz 180 deg; joints [-1.96, -74.915, 109.992, -183.409, 35.125, 182.789]
  MoveL 226 to (-162.16, 850, 50) mm, rotated rx 180 ry 0 rz -180 deg; joints [-3.739, -74.808, 109.852, -186.492, 35.217, 185.312]
  MoveL 227 to (-162.16, 850, -0.5) mm, rotated rx 180 ry 0 rz -180 deg; joints [-3.739, -73.126, 110.672, -186.12, 37.704, 184.849]
  MoveL 228 to (-162.16, 850, 50) mm, rotated rx 180 ry 0 rz -180 deg; joints [-3.739, -74.808, 109.852, -186.492, 35.217, 185.312]
  MoveL 229 to (-162.16, 900, 50) mm, rotated rx -180 ry 0 rz -180 deg; joints [-5.51, -74.636, 109.625, -189.549, 35.366, 187.811]
  MoveL 230 to (-162.16, 900, -0.5) mm, rotated rx -180 ry 0 rz -180 deg; joints [-5.51, -72.958, 110.443, -189.007, 37.829, 187.136]
  MoveL 231 to (-162.16, 900, 50) mm, rotated rx -180 ry 0 rz -180 deg; joints [-5.51, -74.636, 109.625, -189.549, 35.366, 187.811]
  MoveL 232 to (-162.16, 950, 50) mm, rotated rx 180 ry 0 rz -180 deg; joints [-7.27, -74.397, 109.311, -192.566, 35.568, 190.277]
  MoveL 233 to (-162.16, 950, -0.5) mm, rotated rx 180 ry 0 rz -180 deg; joints [-7.27, -72.726, 110.127, -191.862, 37.999, 189.398]
  MoveL 234 to (-162.16, 950, 50) mm, rotated rx 180 ry 0 rz -180 deg; joints [-7.27, -74.397, 109.311, -192.566, 35.568, 190.277]
  MoveL 235 to (-162.16, 1000, 50) mm, rotated rx -180 ry 0 rz -180 deg; joints [-9.017, -74.095, 108.91, -195.534, 35.821, 192.702]
  MoveL 236 to (-162.16, 1000, -0.5) mm, rotated rx 180 ry 0 rz -180 deg; joints [-9.017, -72.432, 109.724, -194.678, 38.212, 191.63]
  MoveL 237 to (-162.16, 1000, 50) mm, rotated rx -180 ry 0 rz -180 deg; joints [-9.017, -74.095, 108.91, -195.534, 35.821, 192.702]
  MoveL 238 to (-162.16, 1050, 50) mm, rotated rx 180 ry 0 rz -180 deg; joints [-10.748, -73.728, 108.422, -198.443, 36.12, 195.077]
  MoveL 239 to (-162.16, 1050, -0.5) mm, rotated rx -180 ry 0 rz -180 deg; joints [-10.748, -72.076, 109.233, -197.446, 38.464, 193.824]
  MoveL 240 to (-162.16, 1050, 50) mm, rotated rx 180 ry 0 rz -180 deg; joints [-10.748, -73.728, 108.422, -198.443, 36.12, 195.077]
  MoveL 241 to (-162.16, 1100, 50) mm, rotated rx -180 ry 0 rz -180 deg; joints [-12.458, -73.3, 107.849, -201.285, 36.462, 197.397]
  MoveL 242 to (-162.16, 1100, -0.5) mm, rotated rx 180 ry 0 rz -180 deg; joints [-12.458, -71.659, 108.657, -200.16, 38.753, 195.977]
  MoveL 243 to (-162.16, 1100, 50) mm, rotated rx -180 ry 0 rz -180 deg; joints [-12.458, -73.3, 107.849, -201.285, 36.462, 197.397]
  MoveL 244 to (-162.16, 1150, 50) mm, rotated rx 180 ry 0 rz 180 deg; joints [-14.147, -72.811, 107.19, -204.054, 36.842, 199.658]
  MoveL 245 to (-162.16, 1150, -0.5) mm, rotated rx 180 ry 0 rz 180 deg; joints [-14.147, -71.183, 107.994, -202.814, 39.074, 198.085]
  MoveL 246 to (-162.16, 1150, 50) mm, rotated rx 180 ry 0 rz 180 deg; joints [-14.147, -72.811, 107.19, -204.054, 36.842, 199.658]
  MoveL 247 to (-162.16, 1200, 50) mm, rotated rx 180 ry 0 rz -180 deg; joints [-15.81, -72.262, 106.446, -206.748, 37.255, 201.858]
  MoveL 248 to (-162.16, 1200, -0.5) mm, rotated rx -180 ry 0 rz -180 deg; joints [-15.81, -70.65, 107.247, -205.406, 39.423, 200.148]
  MoveL 249 to (-162.16, 1200, 50) mm, rotated rx 180 ry 0 rz -180 deg; joints [-15.81, -72.262, 106.446, -206.748, 37.255, 201.858]
  MoveL 250 to (-162.16, 1250, 50) mm, rotated rx -180 ry 0 rz -180 deg; joints [-17.447, -71.656, 105.617, -209.362, 37.697, 203.997]
  MoveL 251 to (-162.16, 1250, -0.5) mm, rotated rx -180 ry 0 rz -180 deg; joints [-17.447, -70.06, 106.414, -207.932, 39.797, 202.163]
  MoveL 252 to (-162.16, 1250, 50) mm, rotated rx -180 ry 0 rz -180 deg; joints [-17.447, -71.656, 105.617, -209.362, 37.697, 203.997]
  MoveL 253 to (-162.16, 1300, 50) mm, rotated rx 180 ry 0 rz -180 deg; joints [-19.055, -70.994, 104.704, -211.896, 38.162, 206.074]
  MoveL 254 to (-162.16, 1300, -0.5) mm, rotated rx 180 ry 0 rz -180 deg; joints [-19.055, -69.415, 105.498, -210.39, 40.192, 204.132]
  MoveL 255 to (-162.16, 1300, 50) mm, rotated rx 180 ry 0 rz -180 deg; joints [-19.055, -70.994, 104.704, -211.896, 38.162, 206.074]
  MoveL 256 to (-162.16, 1350, 50) mm, rotated rx -180 ry 0 rz -180 deg; joints [-20.632, -70.277, 103.708, -214.349, 38.646, 208.092]
  MoveL 257 to (-162.16, 1350, -0.5) mm, rotated rx -180 ry 0 rz -180 deg; joints [-20.632, -68.717, 104.497, -212.78, 40.603, 206.055]
  MoveL 258 to (-162.16, 1350, 50) mm, rotated rx -180 ry 0 rz -180 deg; joints [-20.632, -70.277, 103.708, -214.349, 38.646, 208.092]
  MoveL 259 to (-162.16, 1400, 50) mm, rotated rx 180 ry 0 rz 180 deg; joints [-22.177, -69.508, 102.629, -216.724, 39.144, 210.053]
  MoveL 260 to (-162.16, 1400, -0.5) mm, rotated rx 180 ry 0 rz -180 deg; joints [-22.177, -67.968, 103.414, -215.103, 41.027, 207.935]
  MoveL 261 to (-162.16, 1400, 50) mm, rotated rx 180 ry 0 rz 180 deg; joints [-22.177, -69.508, 102.629, -216.724, 39.144, 210.053]
  MoveL 262 to (-237.84, 50, 50) mm, rotated rx -180 ry 0 rz -180 deg; joints [24.413, -71.775, 105.781, -140.937, 40.987, 148.506]
  MoveL 263 to (-237.84, 50, -0.5) mm, rotated rx -180 ry 0 rz 180 deg; joints [24.413, -70.176, 106.579, -142.59, 42.87, 150.727]
  MoveL 264 to (-237.84, 50, 50) mm, rotated rx -180 ry 0 rz -180 deg; joints [24.413, -71.775, 105.781, -140.937, 40.987, 148.506]
  MoveL 265 to (-237.84, 100, 50) mm, rotated rx -180 ry 0 rz -180 deg; joints [22.843, -72.625, 106.938, -143.23, 40.431, 150.368]
  MoveL 266 to (-237.84, 100, -0.5) mm, rotated rx -180 ry 0 rz -180 deg; joints [22.843, -71.003, 107.742, -144.846, 42.395, 152.522]
  MoveL 267 to (-237.84, 100, 50) mm, rotated rx -180 ry 0 rz -180 deg; joints [22.843, -72.625, 106.938, -143.23, 40.431, 150.368]
  MoveL 268 to (-237.84, 150, 50) mm, rotated rx 180 ry 0 rz -180 deg; joints [21.236, -73.423, 108.013, -145.608, 39.885, 152.29]
  MoveL 269 to (-237.84, 150, -0.5) mm, rotated rx 180 ry 0 rz -180 deg; joints [21.236, -71.779, 108.822, -147.176, 41.929, 154.363]
  MoveL 270 to (-237.84, 150, 50) mm, rotated rx 180 ry 0 rz -180 deg; joints [21.236, -73.423, 108.013, -145.608, 39.885, 152.29]
  MoveL 271 to (-237.84, 200, 50) mm, rotated rx 180 ry 0 rz -180 deg; joints [19.593, -74.167, 109.005, -148.074, 39.354, 154.276]
  MoveL 272 to (-237.84, 200, -0.5) mm, rotated rx -180 ry 0 rz -180 deg; joints [19.593, -72.502, 109.82, -149.581, 41.475, 156.255]
  MoveL 273 to (-237.84, 200, 50) mm, rotated rx 180 ry 0 rz -180 deg; joints [19.593, -74.167, 109.005, -148.074, 39.354, 154.276]
  MoveL 274 to (-237.84, 250, 50) mm, rotated rx 180 ry 0 rz 180 deg; joints [17.915, -74.855, 109.913, -150.629, 38.842, 156.329]
  MoveL 275 to (-237.84, 250, -0.5) mm, rotated rx -180 ry 0 rz -180 deg; joints [17.915, -73.171, 110.733, -152.063, 41.04, 158.199]
  MoveL 276 to (-237.84, 250, 50) mm, rotated rx 180 ry 0 rz 180 deg; joints [17.915, -74.855, 109.913, -150.629, 38.842, 156.329]
  MoveL 277 to (-237.84, 300, 50) mm, rotated rx 180 ry 0 rz -180 deg; joints [16.205, -75.485, 110.737, -153.273, 38.356, 158.453]
  MoveL 278 to (-237.84, 300, -0.5) mm, rotated rx -180 ry 0 rz 180 deg; joints [16.205, -73.783, 111.561, -154.62, 40.626, 160.198]
  MoveL 279 to (-237.84, 300, 50) mm, rotated rx 180 ry 0 rz -180 deg; joints [16.205, -75.485, 110.737, -153.273, 38.356, 158.453]
  MoveL 280 to (-237.84, 350, 50) mm, rotated rx -180 ry 0 rz 180 deg; joints [14.465, -76.054, 111.475, -156.006, 37.9, 160.647]
  MoveL 281 to (-237.84, 350, -0.5) mm, rotated rx -180 ry 0 rz -180 deg; joints [14.465, -74.336, 112.304, -157.251, 40.239, 162.251]
  MoveL 282 to (-237.84, 350, 50) mm, rotated rx -180 ry 0 rz 180 deg; joints [14.465, -76.054, 111.475, -156.006, 37.9, 160.647]
  MoveL 283 to (-237.84, 400, 50) mm, rotated rx 180 ry 0 rz -180 deg; joints [12.698, -76.562, 112.128, -158.824, 37.481, 162.912]
  MoveL 284 to (-237.84, 400, -0.5) mm, rotated rx -180 ry 0 rz -180 deg; joints [12.698, -74.829, 112.961, -159.953, 39.883, 164.357]
  MoveL 285 to (-237.84, 400, 50) mm, rotated rx 180 ry 0 rz -180 deg; joints [12.698, -76.562, 112.128, -158.824, 37.481, 162.912]
  MoveL 286 to (-237.84, 450, 50) mm, rotated rx -180 ry 0 rz -180 deg; joints [10.905, -77.005, 112.693, -161.724, 37.104, 165.244]
  MoveL 287 to (-237.84, 450, -0.5) mm, rotated rx -180 ry 0 rz -180 deg; joints [10.905, -75.259, 113.531, -162.721, 39.564, 166.515]
  MoveL 288 to (-237.84, 450, 50) mm, rotated rx -180 ry 0 rz -180 deg; joints [10.905, -77.005, 112.693, -161.724, 37.104, 165.244]
  MoveL 289 to (-237.84, 500, 50) mm, rotated rx 180 ry 0 rz -180 deg; joints [9.091, -77.382, 113.172, -164.698, 36.776, 167.639]
  MoveL 290 to (-237.84, 500, -0.5) mm, rotated rx 180 ry 0 rz -180 deg; joints [9.091, -75.626, 114.013, -165.551, 39.286, 168.721]
  MoveL 291 to (-237.84, 500, 50) mm, rotated rx 180 ry 0 rz -180 deg; joints [9.091, -77.382, 113.172, -164.698, 36.776, 167.639]
  MoveL 292 to (-237.84, 550, 50) mm, rotated rx 180 ry 0 rz 180 deg; joints [7.258, -77.692, 113.563, -167.738, 36.501, 170.09]
  MoveL 293 to (-237.84, 550, -0.5) mm, rotated rx -180 ry 0 rz 180 deg; joints [7.258, -75.926, 114.406, -168.433, 39.054, 170.969]
  MoveL 294 to (-237.84, 550, 50) mm, rotated rx 180 ry 0 rz 180 deg; joints [7.258, -77.692, 113.563, -167.738, 36.501, 170.09]
  MoveL 295 to (-237.84, 600, 50) mm, rotated rx 180 ry 0 rz 180 deg; joints [5.41, -77.933, 113.865, -170.833, 36.283, 172.588]
  MoveL 296 to (-237.84, 600, -0.5) mm, rotated rx -180 ry 0 rz -180 deg; joints [5.41, -76.16, 114.711, -171.36, 38.87, 173.253]
  MoveL 297 to (-237.84, 600, 50) mm, rotated rx 180 ry 0 rz 180 deg; joints [5.41, -77.933, 113.865, -170.833, 36.283, 172.588]
  MoveL 298 to (-237.84, 650, 50) mm, rotated rx -180 ry 0 rz -180 deg; joints [3.55, -78.104, 114.079, -173.971, 36.126, 175.124]
  MoveL 299 to (-237.84, 650, -0.5) mm, rotated rx -180 ry 0 rz -180 deg; joints [3.55, -76.326, 114.926, -174.321, 38.738, 175.564]
  MoveL 300 to (-237.84, 650, 50) mm, rotated rx -180 ry 0 rz -180 deg; joints [3.55, -78.104, 114.079, -173.971, 36.126, 175.124]
  MoveL 301 to (-237.84, 700, 50) mm, rotated rx -180 ry 0 rz -180 deg; joints [1.683, -78.204, 114.204, -177.138, 36.034, 177.685]
  MoveL 302 to (-237.84, 700, -0.5) mm, rotated rx -180 ry 0 rz -180 deg; joints [1.683, -76.423, 115.052, -177.305, 38.66, 177.895]
  MoveL 303 to (-237.84, 700, 50) mm, rotated rx -180 ry 0 rz -180 deg; joints [1.683, -78.204, 114.204, -177.138, 36.034, 177.685]
  MoveL 304 to (-237.84, 750, 50) mm, rotated rx 180 ry 0 rz -180 deg; joints [-0.187, -78.232, 114.239, -180.318, 36.008, 180.257]
  MoveL 305 to (-237.84, 750, -0.5) mm, rotated rx -180 ry 0 rz -180 deg; joints [-0.187, -76.45, 115.088, -180.3, 38.638, 180.234]
  MoveL 306 to (-237.84, 750, 50) mm, rotated rx 180 ry 0 rz -180 deg; joints [-0.187, -78.232, 114.239, -180.318, 36.008, 180.257]
  MoveL 307 to (-237.84, 800, 50) mm, rotated rx -180 ry 0 rz -180 deg; joints [-2.057, -78.189, 114.186, -183.497, 36.047, 182.829]
  MoveL 308 to (-237.84, 800, -0.5) mm, rotated rx -180 ry 0 rz -180 deg; joints [-2.057, -76.409, 115.034, -183.293, 38.671, 182.572]
  MoveL 309 to (-237.84, 800, 50) mm, rotated rx -180 ry 0 rz -180 deg; joints [-2.057, -78.189, 114.186, -183.497, 36.047, 182.829]
  MoveL 310 to (-237.84, 850, 50) mm, rotated rx -180 ry 0 rz -180 deg; joints [-3.923, -78.075, 114.043, -186.66, 36.153, 185.386]
  MoveL 311 to (-237.84, 850, -0.5) mm, rotated rx 180 ry 0 rz 180 deg; joints [-3.923, -76.298, 114.89, -186.274, 38.76, 184.9]
  MoveL 312 to (-237.84, 850, 50) mm, rotated rx -180 ry 0 rz -180 deg; joints [-3.923, -78.075, 114.043, -186.66, 36.153, 185.386]
  MoveL 313 to (-237.84, 900, 50) mm, rotated rx 180 ry 0 rz 180 deg; joints [-5.78, -77.89, 113.812, -189.79, 36.321, 187.915]
  MoveL 314 to (-237.84, 900, -0.5) mm, rotated rx -180 ry 0 rz -180 deg; joints [-5.78, -76.119, 114.657, -189.229, 38.903, 187.206]
  MoveL 315 to (-237.84, 900, 50) mm, rotated rx 180 ry 0 rz 180 deg; joints [-5.78, -77.89, 113.812, -189.79, 36.321, 187.915]
  MoveL 316 to (-237.84, 950, 50) mm, rotated rx -180 ry 0 rz -180 deg; joints [-7.626, -77.636, 113.492, -192.875, 36.551, 190.405]
  MoveL 317 to (-237.84, 950, -0.5) mm, rotated rx -180 ry 0 rz -180 deg; joints [-7.626, -75.872, 114.334, -192.147, 39.096, 189.484]
  MoveL 318 to (-237.84, 950, 50) mm, rotated rx -180 ry 0 rz -180 deg; joints [-7.626, -77.636, 113.492, -192.875, 36.551, 190.405]
  MoveL 319 to (-237.84, 1000, 50) mm, rotated rx -180 ry 0 rz -180 deg; joints [-9.455, -77.312, 113.083, -195.903, 36.838, 192.845]
  MoveL 320 to (-237.84, 1000, -0.5) mm, rotated rx 180 ry 0 rz -180 deg; joints [-9.455, -75.558, 113.923, -195.02, 39.339, 191.724]
  MoveL 321 to (-237.84, 1000, 50) mm, rotated rx -180 ry 0 rz -180 deg; joints [-9.455, -77.312, 113.083, -195.903, 36.838, 192.845]
  MoveL 322 to (-237.84, 1050, 50) mm, rotated rx -180 ry 0 rz -180 deg; joints [-11.266, -76.922, 112.587, -198.862, 37.176, 195.228]
  MoveL 323 to (-237.84, 1050, -0.5) mm, rotated rx 180 ry 0 rz -180 deg; joints [-11.266, -75.178, 113.424, -197.837, 39.625, 193.92]
  MoveL 324 to (-237.84, 1050, 50) mm, rotated rx -180 ry 0 rz -180 deg; joints [-11.266, -76.922, 112.587, -198.862, 37.176, 195.228]
  MoveL 325 to (-237.84, 1100, 50) mm, rotated rx -180 ry 0 rz -180 deg; joints [-13.053, -76.465, 112.004, -201.746, 37.562, 197.547]
  MoveL 326 to (-237.84, 1100, -0.5) mm, rotated rx -180 ry 0 rz -180 deg; joints [-13.053, -74.735, 112.837, -200.593, 39.952, 196.068]
  MoveL 327 to (-237.84, 1100, 50) mm, rotated rx -180 ry 0 rz -180 deg; joints [-13.053, -76.465, 112.004, -201.746, 37.562, 197.547]
  MoveL 328 to (-237.84, 1150, 50) mm, rotated rx 180 ry 0 rz -180 deg; joints [-14.816, -75.945, 111.334, -204.548, 37.988, 199.797]
  MoveL 329 to (-237.84, 1150, -0.5) mm, rotated rx 180 ry 0 rz 180 deg; joints [-14.816, -74.23, 112.163, -203.281, 40.314, 198.164]
  MoveL 330 to (-237.84, 1150, 50) mm, rotated rx 180 ry 0 rz -180 deg; joints [-14.816, -75.945, 111.334, -204.548, 37.988, 199.797]
  MoveL 331 to (-237.84, 1200, 50) mm, rotated rx 180 ry 0 rz -180 deg; joints [-16.55, -75.363, 110.579, -207.263, 38.451, 201.977]
  MoveL 332 to (-237.84, 1200, -0.5) mm, rotated rx 180 ry 0 rz -180 deg; joints [-16.55, -73.665, 111.403, -205.897, 40.707, 200.206]
  MoveL 333 to (-237.84, 1200, 50) mm, rotated rx 180 ry 0 rz -180 deg; joints [-16.55, -75.363, 110.579, -207.263, 38.451, 201.977]
  MoveL 334 to (-237.84, 1250, 50) mm, rotated rx 180 ry 0 rz 180 deg; joints [-18.253, -74.722, 109.738, -209.889, 38.943, 204.087]
  MoveL 335 to (-237.84, 1250, -0.5) mm, rotated rx 180 ry 0 rz -180 deg; joints [-18.253, -73.041, 110.557, -208.439, 41.125, 202.194]
  MoveL 336 to (-237.84, 1250, 50) mm, rotated rx 180 ry 0 rz 180 deg; joints [-18.253, -74.722, 109.738, -209.889, 38.943, 204.087]
  MoveL 337 to (-237.84, 1300, 50) mm, rotated rx -180 ry 0 rz -180 deg; joints [-19.924, -74.022, 108.814, -212.426, 39.459, 206.127]
  MoveL 338 to (-237.84, 1300, -0.5) mm, rotated rx -180 ry 0 rz -180 deg; joints [-19.924, -72.362, 109.627, -210.906, 41.565, 204.127]
  MoveL 339 to (-237.84, 1300, 50) mm, rotated rx -180 ry 0 rz -180 deg; joints [-19.924, -74.022, 108.814, -212.426, 39.459, 206.127]
  MoveL 340 to (-237.84, 1350, 50) mm, rotated rx 180 ry 0 rz -180 deg; joints [-21.56, -73.267, 107.805, -214.874, 39.993, 208.099]
  MoveL 341 to (-237.84, 1350, -0.5) mm, rotated rx 180 ry 0 rz -180 deg; joints [-21.56, -71.628, 108.613, -213.296, 42.021, 206.009]
  MoveL 342 to (-237.84, 1350, 50) mm, rotated rx 180 ry 0 rz -180 deg; joints [-21.56, -73.267, 107.805, -214.874, 39.993, 208.099]
  MoveL 343 to (-313.52, 50, 50) mm, rotated rx -180 ry 0 rz -180 deg; joints [25.525, -74.696, 109.704, -140.228, 42.343, 148.4]
  MoveL 344 to (-313.52, 50, -0.5) mm, rotated rx 180 ry 0 rz -180 deg; joints [25.525, -73.016, 110.522, -141.894, 44.286, 150.689]
  MoveL 345 to (-313.52, 50, 50) mm, rotated rx -180 ry 0 rz -180 deg; joints [25.525, -74.696, 109.704, -140.228, 42.343, 148.4]
  MoveL 346 to (-313.52, 100, 50) mm, rotated rx -180 ry 0 rz 180 deg; joints [23.901, -75.593, 110.878, -142.505, 41.73, 150.207]
  MoveL 347 to (-313.52, 100, -0.5) mm, rotated rx -180 ry 0 rz -180 deg; joints [23.901, -73.888, 111.703, -144.141, 43.759, 152.434]
  MoveL 348 to (-313.52, 100, 50) mm, rotated rx -180 ry 0 rz 180 deg; joints [23.901, -75.593, 110.878, -142.505, 41.73, 150.207]
  MoveL 349 to (-313.52, 150, 50) mm, rotated rx -180 ry 0 rz -180 deg; joints [22.235, -76.438, 111.969, -144.876, 41.124, 152.081]
  MoveL 350 to (-313.52, 150, -0.5) mm, rotated rx 180 ry 0 rz 180 deg; joints [22.235, -74.709, 112.802, -146.47, 43.24, 154.232]
  MoveL 351 to (-313.52, 150, 50) mm, rotated rx -180 ry 0 rz -180 deg; joints [22.235, -76.438, 111.969, -144.876, 41.124, 152.081]
  MoveL 352 to (-313.52, 200, 50) mm, rotated rx -180 ry 0 rz -180 deg; joints [20.528, -77.229, 112.977, -147.343, 40.531, 154.028]
  MoveL 353 to (-313.52, 200, -0.5) mm, rotated rx 180 ry 0 rz 180 deg; joints [20.528, -75.477, 113.817, -148.884, 42.732, 156.088]
  MoveL 354 to (-313.52, 200, 50) mm, rotated rx -180 ry 0 rz -180 deg; joints [20.528, -77.229, 112.977, -147.343, 40.531, 154.028]
  MoveL 355 to (-313.52, 250, 50) mm, rotated rx 180 ry 0 rz 180 deg; joints [18.783, -77.962, 113.901, -149.91, 39.957, 156.051]
  MoveL 356 to (-313.52, 250, -0.5) mm, rotated rx 180 ry 0 rz 180 deg; joints [18.783, -76.188, 114.747, -151.382, 42.241, 158.005]
  MoveL 357 to (-313.52, 250, 50) mm, rotated rx 180 ry 0 rz 180 deg; joints [18.783, -77.962, 113.901, -149.91, 39.957, 156.051]
  MoveL 358 to (-313.52, 300, 50) mm, rotated rx 180 ry 0 rz 180 deg; joints [17.001, -78.635, 114.74, -152.578, 39.409, 158.155]
  MoveL 359 to (-313.52, 300, -0.5) mm, rotated rx -180 ry 0 rz 180 deg; joints [17.001, -76.841, 115.592, -153.967, 41.773, 159.984]
  MoveL 360 to (-313.52, 300, 50) mm, rotated rx 180 ry 0 rz 180 deg; joints [17.001, -78.635, 114.74, -152.578, 39.409, 158.155]
  MoveL 361 to (-313.52, 350, 50) mm, rotated rx 180 ry 0 rz 180 deg; joints [15.184, -79.245, 115.492, -155.346, 38.893, 160.341]
  MoveL 362 to (-313.52, 350, -0.5) mm, rotated rx 180 ry 0 rz -180 deg; joints [15.184, -77.433, 116.35, -156.635, 41.333, 162.028]
  MoveL 363 to (-313.52, 350, 50) mm, rotated rx 180 ry 0 rz 180 deg; joints [15.184, -79.245, 115.492, -155.346, 38.893, 160.341]
  MoveL 364 to (-313.52, 400, 50) mm, rotated rx 180 ry 0 rz 180 deg; joints [13.335, -79.789, 116.158, -158.212, 38.417, 162.61]
  MoveL 365 to (-313.52, 400, -0.5) mm, rotated rx 180 ry 0 rz 180 deg; joints [13.335, -77.961, 117.021, -159.386, 40.927, 164.134]
  MoveL 366 to (-313.52, 400, 50) mm, rotated rx 180 ry 0 rz 180 deg; joints [13.335, -79.789, 116.158, -158.212, 38.417, 162.61]
  MoveL 367 to (-313.52, 450, 50) mm, rotated rx -180 ry 0 rz -180 deg; joints [11.458, -80.266, 116.735, -161.171, 37.987, 164.957]
  MoveL 368 to (-313.52, 450, -0.5) mm, rotated rx 180 ry 0 rz 180 deg; joints [11.458, -78.423, 117.604, -162.213, 40.561, 166.302]
  MoveL 369 to (-313.52, 450, 50) mm, rotated rx -180 ry 0 rz -180 deg; joints [11.458, -80.266, 116.735, -161.171, 37.987, 164.957]
  MoveL 370 to (-313.52, 500, 50) mm, rotated rx 180 ry 0 rz 180 deg; joints [9.555, -80.672, 117.224, -164.217, 37.611, 167.379]
  MoveL 371 to (-313.52, 500, -0.5) mm, rotated rx -180 ry 0 rz -180 deg; joints [9.555, -78.817, 118.097, -165.111, 40.242, 168.528]
  MoveL 372 to (-313.52, 500, 50) mm, rotated rx 180 ry 0 rz 180 deg; joints [9.555, -80.672, 117.224, -164.217, 37.611, 167.379]
  MoveL 373 to (-313.52, 550, 50) mm, rotated rx 180 ry 0 rz 180 deg; joints [7.631, -81.007, 117.623, -167.34, 37.294, 169.869]
  MoveL 374 to (-313.52, 550, -0.5) mm, rotated rx 180 ry 0 rz 180 deg; joints [7.631, -79.141, 118.499, -168.071, 39.973, 170.804]
  MoveL 375 to (-313.52, 550, 50) mm, rotated rx 180 ry 0 rz 180 deg; joints [7.631, -81.007, 117.623, -167.34, 37.294, 169.869]
  MoveL 376 to (-313.52, 600, 50) mm, rotated rx 180 ry 0 rz 180 deg; joints [5.689, -81.267, 117.933, -170.528, 37.043, 172.415]
  MoveL 377 to (-313.52, 600, -0.5) mm, rotated rx -180 ry 0 rz -180 deg; joints [5.689, -79.393, 118.811, -171.083, 39.761, 173.123]
  MoveL 378 to (-313.52, 600, 50) mm, rotated rx 180 ry 0 rz 180 deg; joints [5.689, -81.267, 117.933, -170.528, 37.043, 172.415]
  MoveL 379 to (-313.52, 650, 50) mm, rotated rx -180 ry 0 rz -180 deg; joints [3.734, -81.451, 118.151, -173.767, 36.863, 175.006]
  MoveL 380 to (-313.52, 650, -0.5) mm, rotated rx 180 ry 0 rz -180 deg; joints [3.734, -79.572, 119.032, -174.136, 39.608, 175.476]
  MoveL 381 to (-313.52, 650, 50) mm, rotated rx -180 ry 0 rz -180 deg; joints [3.734, -81.451, 118.151, -173.767, 36.863, 175.006]
  MoveL 382 to (-313.52, 700, 50) mm, rotated rx -180 ry 0 rz -180 deg; joints [1.771, -81.559, 118.279, -177.04, 36.756, 177.628]
  MoveL 383 to (-313.52, 700, -0.5) mm, rotated rx -180 ry 0 rz -180 deg; joints [1.771, -79.676, 119.161, -177.216, 39.517, 177.852]
  MoveL 384 to (-313.52, 700, 50) mm, rotated rx -180 ry 0 rz -180 deg; joints [1.771, -81.559, 118.279, -177.04, 36.756, 177.628]
  MoveL 385 to (-313.52, 750, 50) mm, rotated rx -180 ry 0 rz -180 deg; joints [-0.197, -81.59, 118.315, -180.329, 36.726, 180.264]
  MoveL 386 to (-313.52, 750, -0.5) mm, rotated rx -180 ry 0 rz -180 deg; joints [-0.197, -79.706, 119.198, -180.309, 39.492, 180.239]
  MoveL 387 to (-313.52, 750, 50) mm, rotated rx -180 ry 0 rz -180 deg; joints [-0.197, -81.59, 118.315, -180.329, 36.726, 180.264]
  MoveL 388 to (-313.52, 800, 50) mm, rotated rx -180 ry 0 rz -180 deg; joints [-2.164, -81.544, 118.261, -183.617, 36.772, 182.898]
  MoveL 389 to (-313.52, 800, -0.5) mm, rotated rx 180 ry 0 rz 180 deg; joints [-2.164, -79.662, 119.142, -183.401, 39.53, 182.625]
  MoveL 390 to (-313.52, 800, 50) mm, rotated rx -180 ry 0 rz -180 deg; joints [-2.164, -81.544, 118.261, -183.617, 36.772, 182.898]
  MoveL 391 to (-313.52, 850, 50) mm, rotated rx -180 ry 0 rz -180 deg; joints [-4.126, -81.42, 118.115, -186.884, 36.893, 185.515]
  MoveL 392 to (-313.52, 850, -0.5) mm, rotated rx -180 ry 0 rz -180 deg; joints [-4.126, -79.542, 118.995, -186.477, 39.633, 184.997]
  MoveL 393 to (-313.52, 850, 50) mm, rotated rx -180 ry 0 rz -180 deg; joints [-4.126, -81.42, 118.115, -186.884, 36.893, 185.515]
  MoveL 394 to (-313.52, 900, 50) mm, rotated rx 180 ry 0 rz -180 deg; joints [-6.079, -81.221, 117.878, -190.114, 37.088, 188.098]
  MoveL 395 to (-313.52, 900, -0.5) mm, rotated rx 180 ry 0 rz 180 deg; joints [-6.079, -79.348, 118.756, -189.523, 39.798, 187.344]
  MoveL 396 to (-313.52, 900, 50) mm, rotated rx 180 ry 0 rz -180 deg; joints [-6.079, -81.221, 117.878, -190.114, 37.088, 188.098]
  MoveL 397 to (-313.52, 950, 50) mm, rotated rx -180 ry 0 rz -180 deg; joints [-8.017, -80.946, 117.551, -193.29, 37.353, 190.634]
  MoveL 398 to (-313.52, 950, -0.5) mm, rotated rx 180 ry 0 rz 180 deg; joints [-8.017, -79.082, 118.426, -192.526, 40.023, 189.655]
  MoveL 399 to (-313.52, 950, 50) mm, rotated rx -180 ry 0 rz -180 deg; joints [-8.017, -80.946, 117.551, -193.29, 37.353, 190.634]
  MoveL 400 to (-313.52, 1000, 50) mm, rotated rx -180 ry 0 rz -180 deg; joints [-9.937, -80.597, 117.134, -196.398, 37.681, 193.111]
  MoveL 401 to (-313.52, 1000, -0.5) mm, rotated rx -180 ry 0 rz -180 deg; joints [-9.937, -78.744, 118.005, -195.474, 40.302, 191.922]
  MoveL 402 to (-313.52, 1000, 50) mm, rotated rx -180 ry 0 rz -180 deg; joints [-9.937, -80.597, 117.134, -196.398, 37.681, 193.111]
  MoveL 403 to (-313.52, 1050, 50) mm, rotated rx 180 ry 0 rz -180 deg; joints [-11.835, -80.176, 116.627, -199.428, 38.069, 195.519]
  MoveL 404 to (-313.52, 1050, -0.5) mm, rotated rx -180 ry 0 rz -180 deg; joints [-11.835, -78.336, 117.494, -198.358, 40.631, 194.136]
  MoveL 405 to (-313.52, 1050, 50) mm, rotated rx 180 ry 0 rz -180 deg; joints [-11.835, -80.176, 116.627, -199.428, 38.069, 195.519]
  MoveL 406 to (-313.52, 1100, 50) mm, rotated rx 180 ry 0 rz -180 deg; joints [-13.707, -79.686, 116.032, -202.369, 38.509, 197.851]
  MoveL 407 to (-313.52, 1100, -0.5) mm, rotated rx 180 ry 0 rz -180 deg; joints [-13.707, -77.86, 116.894, -201.171, 41.005, 196.292]
  MoveL 408 to (-313.52, 1100, 50) mm, rotated rx 180 ry 0 rz -180 deg; joints [-13.707, -79.686, 116.032, -202.369, 38.509, 197.851]
  MoveL 409 to (-313.52, 1150, 50) mm, rotated rx 180 ry 0 rz 180 deg; joints [-15.55, -79.128, 115.349, -205.216, 38.994, 200.102]
  MoveL 410 to (-313.52, 1150, -0.5) mm, rotated rx 180 ry 0 rz -180 deg; joints [-15.55, -77.319, 116.206, -203.905, 41.418, 198.386]
  MoveL 411 to (-313.52, 1150, 50) mm, rotated rx 180 ry 0 rz 180 deg; joints [-15.55, -79.128, 115.349, -205.216, 38.994, 200.102]
  MoveL 412 to (-313.52, 1200, 50) mm, rotated rx 180 ry 0 rz -180 deg; joints [-17.36, -78.505, 114.579, -207.964, 39.517, 202.272]
  MoveL 413 to (-313.52, 1200, -0.5) mm, rotated rx 180 ry 0 rz 180 deg; joints [-17.36, -76.715, 115.43, -206.557, 41.864, 200.417]
  MoveL 414 to (-313.52, 1200, 50) mm, rotated rx 180 ry 0 rz -180 deg; joints [-17.36, -78.505, 114.579, -207.964, 39.517, 202.272]
  MoveL 415 to (-313.52, 1250, 50) mm, rotated rx 180 ry 0 rz 180 deg; joints [-19.135, -77.82, 113.723, -210.611, 40.07, 204.36]
  MoveL 416 to (-313.52, 1250, -0.5) mm, rotated rx 180 ry 0 rz -180 deg; joints [-19.135, -76.05, 114.568, -209.124, 42.338, 202.384]
  MoveL 417 to (-313.52, 1250, 50) mm, rotated rx 180 ry 0 rz 180 deg; joints [-19.135, -77.82, 113.723, -210.611, 40.07, 204.36]
  MoveL 418 to (-313.52, 1300, 50) mm, rotated rx 180 ry 0 rz -180 deg; joints [-20.873, -77.075, 112.782, -213.158, 40.648, 206.368]
  MoveL 419 to (-313.52, 1300, -0.5) mm, rotated rx 180 ry 0 rz -180 deg; joints [-20.873, -75.327, 113.62, -211.606, 42.832, 204.288]
  MoveL 420 to (-313.52, 1300, 50) mm, rotated rx 180 ry 0 rz -180 deg; joints [-20.873, -77.075, 112.782, -213.158, 40.648, 206.368]
  MoveL 421 to (-389.2, 50, 50) mm, rotated rx -180 ry 0 rz 180 deg; joints [26.734, -77.63, 113.484, -139.306, 43.625, 148.098]
  MoveL 422 to (-389.2, 50, -0.5) mm, rotated rx -180 ry 0 rz -180 deg; joints [26.734, -75.866, 114.327, -140.999, 45.627, 150.476]
  MoveL 423 to (-389.2, 50, 50) mm, rotated rx -180 ry 0 rz 180 deg; joints [26.734, -77.63, 113.484, -139.306, 43.625, 148.098]
  MoveL 424 to (-389.2, 100, 50) mm, rotated rx 180 ry 0 rz 180 deg; joints [25.054, -78.585, 114.679, -141.568, 42.943, 149.849]
  MoveL 425 to (-389.2, 100, -0.5) mm, rotated rx -180 ry 0 rz -180 deg; joints [25.054, -76.793, 115.53, -143.239, 45.039, 152.171]
  MoveL 426 to (-389.2, 100, 50) mm, rotated rx 180 ry 0 rz 180 deg; joints [25.054, -78.585, 114.679, -141.568, 42.943, 149.849]
  MoveL 427 to (-389.2, 150, 50) mm, rotated rx -180 ry 0 rz -180 deg; joints [23.327, -79.488, 115.79, -143.932, 42.266, 151.675]
  MoveL 428 to (-389.2, 150, -0.5) mm, rotated rx 180 ry 0 rz -180 deg; joints [23.327, -77.668, 116.651, -145.57, 44.455, 153.928]
  MoveL 429 to (-389.2, 150, 50) mm, rotated rx -180 ry 0 rz -180 deg; joints [23.327, -79.488, 115.79, -143.932, 42.266, 151.675]
  MoveL 430 to (-389.2, 200, 50) mm, rotated rx -180 ry 0 rz -180 deg; joints [21.553, -80.335, 116.818, -146.404, 41.599, 153.583]
  MoveL 431 to (-389.2, 200, -0.5) mm, rotated rx 180 ry 0 rz -180 deg; joints [21.553, -78.489, 117.687, -147.996, 43.881, 155.75]
  MoveL 432 to (-389.2, 200, 50) mm, rotated rx -180 ry 0 rz -180 deg; joints [21.553, -80.335, 116.818, -146.404, 41.599, 153.583]
  MoveL 433 to (-389.2, 250, 50) mm, rotated rx 180 ry 0 rz -180 deg; joints [19.735, -81.122, 117.761, -148.988, 40.95, 155.58]
  MoveL 434 to (-389.2, 250, -0.5) mm, rotated rx 180 ry 0 rz 180 deg; joints [19.735, -79.253, 118.638, -150.517, 43.323, 157.642]
  MoveL 435 to (-389.2, 250, 50) mm, rotated rx 180 ry 0 rz -180 deg; joints [19.735, -81.122, 117.761, -148.988, 40.95, 155.58]
  MoveL 436 to (-389.2, 300, 50) mm, rotated rx -180 ry 0 rz -180 deg; joints [17.875, -81.847, 118.618, -151.686, 40.326, 157.67]
  MoveL 437 to (-389.2, 300, -0.5) mm, rotated rx 180 ry 0 rz 180 deg; joints [17.875, -79.956, 119.503, -153.137, 42.788, 159.609]
  MoveL 438 to (-389.2, 300, 50) mm, rotated rx -180 ry 0 rz -180 deg; joints [17.875, -81.847, 118.618, -151.686, 40.326, 157.67]
  MoveL 439 to (-389.2, 350, 50) mm, rotated rx 180 ry 0 rz -180 deg; joints [15.975, -82.507, 119.388, -154.499, 39.736, 159.856]
  MoveL 440 to (-389.2, 350, -0.5) mm, rotated rx -180 ry 0 rz -180 deg; joints [15.975, -80.594, 120.28, -155.853, 42.282, 161.651]
  MoveL 441 to (-389.2, 350, 50) mm, rotated rx 180 ry 0 rz -180 deg; joints [15.975, -82.507, 119.388, -154.499, 39.736, 159.856]
  MoveL 442 to (-389.2, 400, 50) mm, rotated rx -180 ry 0 rz -180 deg; joints [14.038, -83.097, 120.069, -157.425, 39.189, 162.14]
  MoveL 443 to (-389.2, 400, -0.5) mm, rotated rx 180 ry 0 rz 180 deg; joints [14.038, -81.166, 120.968, -158.664, 41.813, 163.769]
  MoveL 444 to (-389.2, 400, 50) mm, rotated rx -180 ry 0 rz -180 deg; joints [14.038, -83.097, 120.069, -157.425, 39.189, 162.14]
  MoveL 445 to (-389.2, 450, 50) mm, rotated rx 180 ry 0 rz 180 deg; joints [12.068, -83.615, 120.66, -160.461, 38.692, 164.518]
  MoveL 446 to (-389.2, 450, -0.5) mm, rotated rx -180 ry 0 rz -180 deg; joints [12.068, -81.668, 121.565, -161.566, 41.389, 165.96]
  MoveL 447 to (-389.2, 450, 50) mm, rotated rx 180 ry 0 rz 180 deg; joints [12.068, -83.615, 120.66, -160.461, 38.692, 164.518]
  MoveL 448 to (-389.2, 500, 50) mm, rotated rx 180 ry 0 rz -180 deg; joints [10.069, -84.057, 121.161, -163.599, 38.256, 166.986]
  MoveL 449 to (-389.2, 500, -0.5) mm, rotated rx -180 ry 0 rz 180 deg; joints [10.069, -82.096, 122.072, -164.55, 41.017, 168.221]
  MoveL 450 to (-389.2, 500, 50) mm, rotated rx 180 ry 0 rz -180 deg; joints [10.069, -84.057, 121.161, -163.599, 38.256, 166.986]
  MoveL 451 to (-389.2, 550, 50) mm, rotated rx 180 ry 0 rz 180 deg; joints [8.044, -84.421, 121.571, -166.829, 37.887, 169.536]
  MoveL 452 to (-389.2, 550, -0.5) mm, rotated rx -180 ry 0 rz -180 deg; joints [8.044, -82.449, 122.485, -167.609, 40.703, 170.544]
  MoveL 453 to (-389.2, 550, 50) mm, rotated rx 180 ry 0 rz 180 deg; joints [8.044, -84.421, 121.571, -166.829, 37.887, 169.536]
  MoveL 454 to (-389.2, 600, 50) mm, rotated rx -180 ry 0 rz -180 deg; joints [5.999, -84.705, 121.888, -170.136, 37.594, 172.155]
  MoveL 455 to (-389.2, 600, -0.5) mm, rotated rx 180 ry 0 rz 180 deg; joints [5.999, -82.724, 122.806, -170.731, 40.454, 172.921]
  MoveL 456 to (-389.2, 600, 50) mm, rotated rx -180 ry 0 rz -180 deg; joints [5.999, -84.705, 121.888, -170.136, 37.594, 172.155]
  MoveL 457 to (-389.2, 650, 50) mm, rotated rx -180 ry 0 rz -180 deg; joints [3.939, -84.907, 122.112, -173.504, 37.383, 174.83]
  MoveL 458 to (-389.2, 650, -0.5) mm, rotated rx -180 ry 0 rz 180 deg; joints [3.939, -82.919, 123.033, -173.901, 40.274, 175.339]
  MoveL 459 to (-389.2, 650, 50) mm, rotated rx -180 ry 0 rz -180 deg; joints [3.939, -84.907, 122.112, -173.504, 37.383, 174.83]
  MoveL 460 to (-389.2, 700, 50) mm, rotated rx 180 ry 0 rz 180 deg; joints [1.868, -85.025, 122.243, -176.914, 37.258, 177.543]
  MoveL 461 to (-389.2, 700, -0.5) mm, rotated rx 180 ry 0 rz -180 deg; joints [1.868, -83.033, 123.165, -177.103, 40.168, 177.786]
  MoveL 462 to (-389.2, 700, 50) mm, rotated rx 180 ry 0 rz 180 deg; joints [1.868, -85.025, 122.243, -176.914, 37.258, 177.543]
  MoveL 463 to (-389.2, 750, 50) mm, rotated rx -180 ry 0 rz -180 deg; joints [-0.208, -85.059, 122.281, -180.343, 37.222, 180.273]
  MoveL 464 to (-389.2, 750, -0.5) mm, rotated rx -180 ry 0 rz -180 deg; joints [-0.208, -83.066, 123.203, -180.322, 40.138, 180.246]
  MoveL 465 to (-389.2, 750, 50) mm, rotated rx -180 ry 0 rz -180 deg; joints [-0.208, -85.059, 122.281, -180.343, 37.222, 180.273]
  MoveL 466 to (-389.2, 800, 50) mm, rotated rx 180 ry 0 rz -180 deg; joints [-2.283, -85.008, 122.224, -183.771, 37.276, 183.002]
  MoveL 467 to (-389.2, 800, -0.5) mm, rotated rx -180 ry 0 rz -180 deg; joints [-2.283, -83.017, 123.146, -183.539, 40.183, 182.705]
  MoveL 468 to (-389.2, 800, 50) mm, rotated rx 180 ry 0 rz -180 deg; joints [-2.283, -85.008, 122.224, -183.771, 37.276, 183.002]
  MoveL 469 to (-389.2, 850, 50) mm, rotated rx -180 ry 0 rz -180 deg; joints [-4.352, -84.873, 122.075, -187.174, 37.418, 185.708]
  MoveL 470 to (-389.2, 850, -0.5) mm, rotated rx -180 ry 0 rz -180 deg; joints [-4.352, -82.886, 122.995, -186.737, 40.305, 185.147]
  MoveL 471 to (-389.2, 850, 50) mm, rotated rx -180 ry 0 rz -180 deg; joints [-4.352, -84.873, 122.075, -187.174, 37.418, 185.708]
  MoveL 472 to (-389.2, 900, 50) mm, rotated rx 180 ry 0 rz 180 deg; joints [-6.409, -84.655, 121.832, -190.531, 37.646, 188.374]
  MoveL 473 to (-389.2, 900, -0.5) mm, rotated rx 180 ry 0 rz -180 deg; joints [-6.409, -82.675, 122.749, -189.898, 40.498, 187.558]
  MoveL 474 to (-389.2, 900, 50) mm, rotated rx 180 ry 0 rz 180 deg; joints [-6.409, -84.655, 121.832, -190.531, 37.646, 188.374]
  MoveL 475 to (-389.2, 950, 50) mm, rotated rx 180 ry 0 rz 180 deg; joints [-8.451, -84.355, 121.496, -193.824, 37.955, 190.98]
  MoveL 476 to (-389.2, 950, -0.5) mm, rotated rx 180 ry 0 rz -180 deg; joints [-8.451, -82.384, 122.41, -193.008, 40.761, 189.925]
  MoveL 477 to (-389.2, 950, 50) mm, rotated rx 180 ry 0 rz 180 deg; joints [-8.451, -84.355, 121.496, -193.824, 37.955, 190.98]
  MoveL 478 to (-389.2, 1000, 50) mm, rotated rx -180 ry 0 rz -180 deg; joints [-10.471, -83.975, 121.068, -197.036, 38.338, 193.515]
  MoveL 479 to (-389.2, 1000, -0.5) mm, rotated rx 180 ry 0 rz -180 deg; joints [-10.471, -82.016, 121.978, -196.053, 41.087, 192.237]
  MoveL 480 to (-389.2, 1000, 50) mm, rotated rx -180 ry 0 rz -180 deg; joints [-10.471, -83.975, 121.068, -197.036, 38.338, 193.515]
  MoveL 481 to (-389.2, 1050, 50) mm, rotated rx 180 ry 0 rz 180 deg; joints [-12.465, -83.517, 120.549, -200.154, 38.787, 195.965]
  MoveL 482 to (-389.2, 1050, -0.5) mm, rotated rx -180 ry 0 rz -180 deg; joints [-12.465, -81.573, 121.453, -199.021, 41.47, 194.484]
  MoveL 483 to (-389.2, 1050, 50) mm, rotated rx 180 ry 0 rz 180 deg; joints [-12.465, -83.517, 120.549, -200.154, 38.787, 195.965]
  MoveL 484 to (-389.2, 1100, 50) mm, rotated rx -180 ry 0 rz -180 deg; joints [-14.428, -82.985, 119.94, -203.169, 39.294, 198.325]
  MoveL 485 to (-389.2, 1100, -0.5) mm, rotated rx -180 ry 0 rz -180 deg; joints [-14.428, -81.057, 120.837, -201.905, 41.904, 196.661]
  MoveL 486 to (-389.2, 1100, 50) mm, rotated rx -180 ry 0 rz -180 deg; joints [-14.428, -82.985, 119.94, -203.169, 39.294, 198.325]
  MoveL 487 to (-389.2, 1150, 50) mm, rotated rx -180 ry 0 rz 180 deg; joints [-16.358, -82.38, 119.241, -206.073, 39.851, 200.589]
  MoveL 488 to (-389.2, 1150, -0.5) mm, rotated rx 180 ry 0 rz -180 deg; joints [-16.358, -80.472, 120.132, -204.698, 42.38, 198.764]
  MoveL 489 to (-389.2, 1150, 50) mm, rotated rx -180 ry 0 rz 180 deg; joints [-16.358, -82.38, 119.241, -206.073, 39.851, 200.589]
  MoveL 490 to (-389.2, 1200, 50) mm, rotated rx -180 ry 0 rz -180 deg; joints [-18.25, -81.708, 118.454, -208.863, 40.449, 202.755]
  MoveL 491 to (-389.2, 1200, -0.5) mm, rotated rx 180 ry 0 rz -180 deg; joints [-18.25, -79.82, 119.337, -207.395, 42.893, 200.791]
  MoveL 492 to (-389.2, 1200, 50) mm, rotated rx -180 ry 0 rz -180 deg; joints [-18.25, -81.708, 118.454, -208.863, 40.449, 202.755]
  MoveL 493 to (-33.64, 230, 50) mm, rotated rx 180 ry 0 rz 180 deg; joints [16.529, -66.353, 98.098, -150.575, 35.388, 155.305]
  MoveL 494 to (-33.64, 230, -0.5) mm, rotated rx 180 ry 0 rz 180 deg; joints [16.529, -64.892, 98.87, -152.031, 37.346, 157.113]
  MoveL 495 to (-33.64, 230, 50) mm, rotated rx 180 ry 0 rz 180 deg; joints [16.529, -66.353, 98.098, -150.575, 35.388, 155.305]
  MoveL 496 to (-63.64, 230, 50) mm, rotated rx -180 ry 0 rz -180 deg; joints [16.804, -67.563, 99.855, -150.522, 35.978, 155.419]
  MoveL 497 to (-63.64, 230, -0.5) mm, rotated rx -180 ry 0 rz -180 deg; joints [16.804, -66.072, 100.631, -151.97, 37.965, 157.231]
  MoveL 498 to (-63.64, 230, 50) mm, rotated rx -180 ry 0 rz -180 deg; joints [16.804, -67.563, 99.855, -150.522, 35.978, 155.419]
  MoveL 499 to (-109.34, 230, 50) mm, rotated rx 180 ry 0 rz 180 deg; joints [17.239, -69.402, 102.479, -150.379, 36.842, 155.534]
  MoveL 500 to (-109.34, 230, -0.5) mm, rotated rx -180 ry 0 rz -180 deg; joints [17.239, -67.865, 103.264, -151.823, 38.875, 157.362]
  MoveL 501 to (-109.34, 230, 50) mm, rotated rx 180 ry 0 rz 180 deg; joints [17.239, -69.402, 102.479, -150.379, 36.842, 155.534]
  MoveL 502 to (-139.34, 230, 50) mm, rotated rx 180 ry 0 rz 180 deg; joints [17.537, -70.609, 104.171, -150.246, 37.386, 155.573]
  MoveL 503 to (-139.34, 230, -0.5) mm, rotated rx 180 ry 0 rz 180 deg; joints [17.537, -69.041, 104.962, -151.69, 39.45, 157.415]
  MoveL 504 to (-139.34, 230, 50) mm, rotated rx 180 ry 0 rz 180 deg; joints [17.537, -70.609, 104.171, -150.246, 37.386, 155.573]
  MoveL 505 to (-185.04, 230, 50) mm, rotated rx -180 ry 0 rz -180 deg; joints [18.011, -72.45, 106.702, -149.986, 38.18, 155.577]
  MoveL 506 to (-185.04, 230, -0.5) mm, rotated rx -180 ry 0 rz -180 deg; joints [18.011, -70.833, 107.504, -151.436, 40.291, 157.449]
  MoveL 507 to (-185.04, 230, 50) mm, rotated rx -180 ry 0 rz -180 deg; joints [18.011, -72.45, 106.702, -149.986, 38.18, 155.577]
  MoveL 508 to (-215.04, 230, 50) mm, rotated rx 180 ry 0 rz 180 deg; joints [18.336, -73.663, 108.334, -149.776, 38.678, 155.544]
  MoveL 509 to (-215.04, 230, -0.5) mm, rotated rx 180 ry 0 rz -180 deg; joints [18.336, -72.012, 109.145, -151.233, 40.821, 157.439]
  MoveL 510 to (-215.04, 230, 50) mm, rotated rx 180 ry 0 rz 180 deg; joints [18.336, -73.663, 108.334, -149.776, 38.678, 155.544]
  MoveL 511 to (-260.74, 230, 50) mm, rotated rx 180 ry 0 rz -180 deg; joints [18.853, -75.517, 110.779, -149.398, 39.401, 155.438]
  MoveL 512 to (-260.74, 230, -0.5) mm, rotated rx -180 ry 0 rz 180 deg; joints [18.853, -73.814, 111.604, -150.872, 41.594, 157.377]
  MoveL 513 to (-260.74, 230, 50) mm, rotated rx 180 ry 0 rz -180 deg; joints [18.853, -75.517, 110.779, -149.398, 39.401, 155.438]
  MoveL 514 to (-290.74, 230, 50) mm, rotated rx 180 ry 0 rz -180 deg; joints [19.207, -76.741, 112.357, -149.11, 39.853, 155.333]
  MoveL 515 to (-290.74, 230, -0.5) mm, rotated rx 180 ry 0 rz 180 deg; joints [19.207, -75.003, 113.192, -150.599, 42.079, 157.303]
  MoveL 516 to (-290.74, 230, 50) mm, rotated rx 180 ry 0 rz -180 deg; joints [19.207, -76.741, 112.357, -149.11, 39.853, 155.333]
  MoveL 517 to (-336.44, 230, 50) mm, rotated rx 180 ry 0 rz 180 deg; joints [19.773, -78.62, 114.722, -148.612, 40.506, 155.114]
  MoveL 518 to (-336.44, 230, -0.5) mm, rotated rx -180 ry 0 rz 180 deg; joints [19.773, -76.827, 115.574, -150.128, 42.783, 157.142]
  MoveL 519 to (-336.44, 230, 50) mm, rotated rx 180 ry 0 rz 180 deg; joints [19.773, -78.62, 114.722, -148.612, 40.506, 155.114]
  MoveL 520 to (-366.44, 230, 50) mm, rotated rx 180 ry 0 rz 180 deg; joints [20.163, -79.864, 116.249, -148.243, 40.912, 154.931]
  MoveL 521 to (-366.44, 230, -0.5) mm, rotated rx -180 ry 0 rz -180 deg; joints [20.163, -78.033, 117.113, -149.781, 43.223, 157.002]
  MoveL 522 to (-366.44, 230, 50) mm, rotated rx 180 ry 0 rz 180 deg; joints [20.163, -79.864, 116.249, -148.243, 40.912, 154.931]
  MoveL 523 to (-33.64, 420, 50) mm, rotated rx -180 ry 0 rz 180 deg; joints [10.608, -68.231, 100.815, -160.824, 34.085, 163.933]
  MoveL 524 to (-33.64, 420, -0.5) mm, rotated rx 180 ry 0 rz 180 deg; joints [10.608, -66.724, 101.594, -161.863, 36.252, 165.203]
  MoveL 525 to (-33.64, 420, 50) mm, rotated rx -180 ry 0 rz 180 deg; joints [10.608, -68.231, 100.815, -160.824, 34.085, 163.933]
  MoveL 526 to (-63.64, 420, 50) mm, rotated rx 180 ry 0 rz 180 deg; joints [10.79, -69.472, 102.579, -160.765, 34.629, 163.981]
  MoveL 527 to (-63.64, 420, -0.5) mm, rotated rx 180 ry 0 rz 180 deg; joints [10.79, -67.934, 103.364, -161.802, 36.83, 165.258]
  MoveL 528 to (-63.64, 420, 50) mm, rotated rx 180 ry 0 rz 180 deg; joints [10.79, -69.472, 102.579, -160.765, 34.629, 163.981]
  MoveL 529 to (-109.34, 420, 50) mm, rotated rx -180 ry 0 rz -180 deg; joints [11.08, -71.366, 105.218, -160.632, 35.413, 164.013]
  MoveL 530 to (-109.34, 420, -0.5) mm, rotated rx -180 ry 0 rz -180 deg; joints [11.08, -69.778, 106.014, -161.671, 37.669, 165.307]
  MoveL 531 to (-109.34, 420, 50) mm, rotated rx -180 ry 0 rz -180 deg; joints [11.08, -71.366, 105.218, -160.632, 35.413, 164.013]
  MoveL 532 to (-139.34, 420, 50) mm, rotated rx -180 ry 0 rz 180 deg; joints [11.278, -72.613, 106.922, -160.516, 35.898, 164.007]
  MoveL 533 to (-139.34, 420, -0.5) mm, rotated rx 180 ry 0 rz 180 deg; joints [11.278, -70.991, 107.725, -161.56, 38.192, 165.315]
  MoveL 534 to (-139.34, 420, 50) mm, rotated rx -180 ry 0 rz 180 deg; joints [11.278, -72.613, 106.922, -160.516, 35.898, 164.007]
  MoveL 535 to (-185.04, 420, 50) mm, rotated rx 180 ry 0 rz -180 deg; joints [11.595, -74.522, 109.475, -160.295, 36.593, 163.957]
  MoveL 536 to (-185.04, 420, -0.5) mm, rotated rx 180 ry 0 rz 180 deg; joints [11.595, -72.847, 110.292, -161.352, 38.946, 165.294]
  MoveL 537 to (-185.04, 420, 50) mm, rotated rx 180 ry 0 rz -180 deg; joints [11.595, -74.522, 109.475, -160.295, 36.593, 163.957]
  MoveL 538 to (-215.04, 420, 50) mm, rotated rx 180 ry 0 rz -180 deg; joints [11.813, -75.783, 111.124, -160.122, 37.018, 163.897]
  MoveL 539 to (-215.04, 420, -0.5) mm, rotated rx 180 ry 0 rz -180 deg; joints [11.813, -74.073, 111.951, -161.19, 39.412, 165.256]
  MoveL 540 to (-215.04, 420, 50) mm, rotated rx 180 ry 0 rz -180 deg; joints [11.813, -75.783, 111.124, -160.122, 37.018, 163.897]
  MoveL 541 to (-260.74, 420, 50) mm, rotated rx 180 ry 0 rz 180 deg; joints [12.16, -77.72, 113.598, -159.813, 37.619, 163.763]
  MoveL 542 to (-260.74, 420, -0.5) mm, rotated rx 180 ry 0 rz -180 deg; joints [12.16, -75.954, 114.442, -160.902, 40.077, 165.162]
  MoveL 543 to (-260.74, 420, 50) mm, rotated rx 180 ry 0 rz 180 deg; joints [12.16, -77.72, 113.598, -159.813, 37.619, 163.763]
  MoveL 544 to (-290.74, 420, 50) mm, rotated rx -180 ry 0 rz -180 deg; joints [12.399, -79.005, 115.198, -159.579, 37.981, 163.645]
  MoveL 545 to (-290.74, 420, -0.5) mm, rotated rx -180 ry 0 rz -180 deg; joints [12.399, -77.2, 116.053, -160.686, 40.484, 165.074]
  MoveL 546 to (-290.74, 420, 50) mm, rotated rx -180 ry 0 rz -180 deg; joints [12.399, -79.005, 115.198, -159.579, 37.981, 163.645]
  MoveL 547 to (-336.44, 420, 50) mm, rotated rx 180 ry 0 rz 180 deg; joints [12.782, -80.985, 117.598, -159.174, 38.483, 163.418]
  MoveL 548 to (-336.44, 420, -0.5) mm, rotated rx -180 ry 0 rz 180 deg; joints [12.782, -79.12, 118.474, -160.314, 41.055, 164.902]
  MoveL 549 to (-336.44, 420, 50) mm, rotated rx 180 ry 0 rz 180 deg; joints [12.782, -80.985, 117.598, -159.174, 38.483, 163.418]
  MoveL 550 to (-366.44, 420, 50) mm, rotated rx 180 ry 0 rz 180 deg; joints [13.046, -82.303, 119.15, -158.874, 38.778, 163.236]
  MoveL 551 to (-366.44, 420, -0.5) mm, rotated rx -180 ry 0 rz -180 deg; joints [13.046, -80.397, 120.04, -160.039, 41.397, 164.76]
  MoveL 552 to (-366.44, 420, 50) mm, rotated rx 180 ry 0 rz 180 deg; joints [13.046, -82.303, 119.15, -158.874, 38.778, 163.236]
  MoveL 553 to (-33.64, 730, 50) mm, rotated rx 180 ry 0 rz 180 deg; joints [0.495, -69.499, 102.616, -179.094, 33.121, 179.241]
  MoveL 554 to (-33.64, 730, -0.5) mm, rotated rx 180 ry 0 rz 180 deg; joints [0.495, -67.959, 103.401, -179.146, 35.445, 179.304]
  MoveL 555 to (-33.64, 730, 50) mm, rotated rx 180 ry 0 rz 180 deg; joints [0.495, -69.499, 102.616, -179.094, 33.121, 179.241]
  MoveL 556 to (-63.64, 730, 50) mm, rotated rx -180 ry 0 rz 180 deg; joints [0.504, -70.764, 104.386, -179.09, 33.625, 179.242]
  MoveL 557 to (-63.64, 730, -0.5) mm, rotated rx 180 ry 0 rz 180 deg; joints [0.504, -69.192, 105.178, -179.142, 35.99, 179.306]
  MoveL 558 to (-63.64, 730, 50) mm, rotated rx -180 ry 0 rz 180 deg; joints [0.504, -70.764, 104.386, -179.09, 33.625, 179.242]
  MoveL 559 to (-109.34, 730, 50) mm, rotated rx 180 ry 0 rz 180 deg; joints [0.518, -72.699, 107.038, -179.082, 34.343, 179.242]
  MoveL 560 to (-109.34, 730, -0.5) mm, rotated rx -180 ry 0 rz -180 deg; joints [0.518, -71.075, 107.842, -179.135, 36.771, 179.307]
  MoveL 561 to (-109.34, 730, 50) mm, rotated rx 180 ry 0 rz 180 deg; joints [0.518, -72.699, 107.038, -179.082, 34.343, 179.242]
  MoveL 562 to (-139.34, 730, 50) mm, rotated rx -180 ry 0 rz -180 deg; joints [0.527, -73.976, 108.752, -179.075, 34.779, 179.241]
  MoveL 563 to (-139.34, 730, -0.5) mm, rotated rx 180 ry 0 rz 180 deg; joints [0.527, -72.317, 109.565, -179.129, 37.252, 179.306]
  MoveL 564 to (-139.34, 730, 50) mm, rotated rx -180 ry 0 rz -180 deg; joints [0.527, -73.976, 108.752, -179.075, 34.779, 179.241]
  MoveL 565 to (-185.04, 730, 50) mm, rotated rx -180 ry 0 rz 180 deg; joints [0.543, -75.936, 111.322, -179.063, 35.39, 179.236]
  MoveL 566 to (-185.04, 730, -0.5) mm, rotated rx 180 ry 0 rz -180 deg; joints [0.543, -74.221, 112.151, -179.117, 37.933, 179.304]
  MoveL 567 to (-185.04, 730, 50) mm, rotated rx -180 ry 0 rz 180 deg; joints [0.543, -75.936, 111.322, -179.063, 35.39, 179.236]
  MoveL 568 to (-215.04, 730, 50) mm, rotated rx 180 ry 0 rz -180 deg; joints [0.553, -77.235, 112.985, -179.053, 35.754, 179.232]
  MoveL 569 to (-215.04, 730, -0.5) mm, rotated rx -180 ry 0 rz -180 deg; joints [0.553, -75.482, 113.824, -179.109, 38.345, 179.301]
  MoveL 570 to (-215.04, 730, 50) mm, rotated rx 180 ry 0 rz -180 deg; joints [0.553, -77.235, 112.985, -179.053, 35.754, 179.232]
  MoveL 571 to (-260.74, 730, 50) mm, rotated rx -180 ry 0 rz -180 deg; joints [0.57, -79.236, 115.481, -179.036, 36.249, 179.223]
  MoveL 572 to (-260.74, 730, -0.5) mm, rotated rx 180 ry 0 rz -180 deg; joints [0.57, -77.424, 116.339, -179.093, 38.919, 179.294]
  MoveL 573 to (-260.74, 730, 50) mm, rotated rx -180 ry 0 rz -180 deg; joints [0.57, -79.236, 115.481, -179.036, 36.249, 179.223]
  MoveL 574 to (-290.74, 730, 50) mm, rotated rx 180 ry 0 rz 180 deg; joints [0.581, -80.566, 117.097, -179.023, 36.535, 179.215]
  MoveL 575 to (-290.74, 730, -0.5) mm, rotated rx -180 ry 0 rz -180 deg; joints [0.581, -78.714, 117.968, -179.081, 39.258, 179.289]
  MoveL 576 to (-290.74, 730, 50) mm, rotated rx 180 ry 0 rz 180 deg; joints [0.581, -80.566, 117.097, -179.023, 36.535, 179.215]
  MoveL 577 to (-336.44, 730, 50) mm, rotated rx 180 ry 0 rz 180 deg; joints [0.6, -82.624, 119.524, -179.001, 36.904, 179.201]
  MoveL 578 to (-336.44, 730, -0.5) mm, rotated rx -180 ry 0 rz -180 deg; joints [0.6, -80.708, 120.418, -179.061, 39.713, 179.278]
  MoveL 579 to (-336.44, 730, 50) mm, rotated rx 180 ry 0 rz 180 deg; joints [0.6, -82.624, 119.524, -179.001, 36.904, 179.201]
  MoveL 580 to (-366.44, 730, 50) mm, rotated rx 180 ry 0 rz 180 deg; joints [0.613, -83.999, 121.096, -178.984, 37.101, 179.19]
  MoveL 581 to (-366.44, 730, -0.5) mm, rotated rx 180 ry 0 rz 180 deg; joints [0.613, -82.04, 122.005, -179.046, 39.97, 179.269]
  MoveL 582 to (-366.44, 730, 50) mm, rotated rx 180 ry 0 rz 180 deg; joints [0.613, -83.999, 121.096, -178.984, 37.101, 179.19]
  MoveL 583 to (-33.64, 1020, 50) mm, rotated rx -180 ry 0 rz -180 deg; joints [-9.005, -68.59, 101.327, -196.332, 33.82, 193.682]
  MoveL 584 to (-33.64, 1020, -0.5) mm, rotated rx 180 ry 0 rz 180 deg; joints [-9.005, -67.073, 102.108, -195.432, 36.029, 192.584]
  MoveL 585 to (-33.64, 1020, 50) mm, rotated rx -180 ry 0 rz -180 deg; joints [-9.005, -68.59, 101.327, -196.332, 33.82, 193.682]
  MoveL 586 to (-63.64, 1020, 50) mm, rotated rx 180 ry 0 rz -180 deg; joints [-9.16, -69.837, 103.092, -196.387, 34.353, 193.646]
  MoveL 587 to (-63.64, 1020, -0.5) mm, rotated rx 180 ry 0 rz -180 deg; joints [-9.16, -68.289, 103.879, -195.487, 36.599, 192.541]
  MoveL 588 to (-63.64, 1020, 50) mm, rotated rx 180 ry 0 rz -180 deg; joints [-9.16, -69.837, 103.092, -196.387, 34.353, 193.646]
  MoveL 589 to (-109.34, 1020, 50) mm, rotated rx -180 ry 0 rz -180 deg; joints [-9.408, -71.742, 105.735, -196.508, 35.12, 193.626]
  MoveL 590 to (-109.34, 1020, -0.5) mm, rotated rx -180 ry 0 rz -180 deg; joints [-9.408, -70.144, 106.533, -195.605, 37.423, 192.506]
  MoveL 591 to (-109.34, 1020, 50) mm, rotated rx -180 ry 0 rz -180 deg; joints [-9.408, -71.742, 105.735, -196.508, 35.12, 193.626]
  MoveL 592 to (-139.34, 1020, 50) mm, rotated rx 180 ry 0 rz 180 deg; joints [-9.578, -72.997, 107.442, -196.612, 35.592, 193.637]
  MoveL 593 to (-139.34, 1020, -0.5) mm, rotated rx -180 ry 0 rz -180 deg; joints [-9.578, -71.365, 108.248, -195.704, 37.934, 192.503]
  MoveL 594 to (-139.34, 1020, 50) mm, rotated rx 180 ry 0 rz 180 deg; joints [-9.578, -72.997, 107.442, -196.612, 35.592, 193.637]
  MoveL 595 to (-185.04, 1020, 50) mm, rotated rx 180 ry 0 rz -180 deg; joints [-9.849, -74.92, 109.999, -196.809, 36.264, 193.689]
  MoveL 596 to (-185.04, 1020, -0.5) mm, rotated rx -180 ry 0 rz -180 deg; joints [-9.849, -73.234, 110.82, -195.889, 38.669, 192.53]
  MoveL 597 to (-185.04, 1020, 50) mm, rotated rx 180 ry 0 rz -180 deg; joints [-9.849, -74.92, 109.999, -196.809, 36.264, 193.689]
  MoveL 598 to (-215.04, 1020, 50) mm, rotated rx 180 ry 0 rz -180 deg; joints [-10.036, -76.192, 111.652, -196.964, 36.673, 193.748]
  MoveL 599 to (-215.04, 1020, -0.5) mm, rotated rx -180 ry 0 rz 180 deg; joints [-10.036, -74.47, 112.483, -196.032, 39.121, 192.568]
  MoveL 600 to (-215.04, 1020, 50) mm, rotated rx 180 ry 0 rz -180 deg; joints [-10.036, -76.192, 111.652, -196.964, 36.673, 193.748]
  MoveL 601 to (-260.74, 1020, 50) mm, rotated rx 180 ry 0 rz -180 deg; joints [-10.333, -78.147, 114.132, -197.239, 37.246, 193.875]
  MoveL 602 to (-260.74, 1020, -0.5) mm, rotated rx -180 ry 0 rz 180 deg; joints [-10.333, -76.367, 114.98, -196.287, 39.762, 192.658]
  MoveL 603 to (-260.74, 1020, 50) mm, rotated rx 180 ry 0 rz -180 deg; joints [-10.333, -78.147, 114.132, -197.239, 37.246, 193.875]
  MoveL 604 to (-290.74, 1020, 50) mm, rotated rx 180 ry 0 rz 180 deg; joints [-10.538, -79.444, 115.736, -197.447, 37.589, 193.985]
  MoveL 605 to (-290.74, 1020, -0.5) mm, rotated rx 180 ry 0 rz -180 deg; joints [-10.538, -77.626, 116.596, -196.478, 40.15, 192.74]
  MoveL 606 to (-290.74, 1020, 50) mm, rotated rx 180 ry 0 rz 180 deg; joints [-10.538, -79.444, 115.736, -197.447, 37.589, 193.985]
  MoveL 607 to (-336.44, 1020, 50) mm, rotated rx 180 ry 0 rz -180 deg; joints [-10.867, -81.445, 118.144, -197.808, 38.056, 194.194]
  MoveL 608 to (-336.44, 1020, -0.5) mm, rotated rx -180 ry 0 rz -180 deg; joints [-10.867, -79.566, 119.024, -196.807, 40.691, 192.9]
  MoveL 609 to (-336.44, 1020, 50) mm, rotated rx 180 ry 0 rz -180 deg; joints [-10.867, -81.445, 118.144, -197.808, 38.056, 194.194]
  MoveL 610 to (-366.44, 1020, 50) mm, rotated rx 180 ry 0 rz 180 deg; joints [-11.093, -82.778, 119.702, -198.075, 38.326, 194.362]
  MoveL 611 to (-366.44, 1020, -0.5) mm, rotated rx 180 ry 0 rz -180 deg; joints [-11.093, -80.857, 120.597, -197.05, 41.011, 193.03]
  MoveL 612 to (-366.44, 1020, 50) mm, rotated rx 180 ry 0 rz 180 deg; joints [-11.093, -82.778, 119.702, -198.075, 38.326, 194.362]
  Set speed (1000.0 mm/s)
  MoveL 613 to (-366.44, 1020, 50) mm, rotated rx 180 ry 0 rz 180 deg; joints [-11.093, -82.778, 119.702, -198.075, 38.326, 194.362]
  MoveL 614 to (-366.44, 1020, 150) mm, rotated rx -180 ry 0 rz -180 deg; joints [-11.093, -86.191, 117.594, -200.621, 33.115, 197.494]
